ABB RAPID module: P454.mod

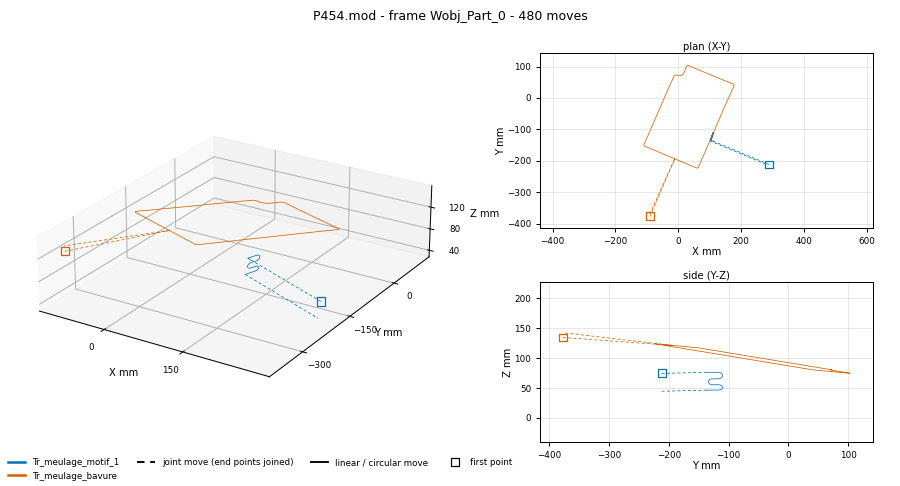
[picture p0: tool path of P454.mod in frame Wobj_Part_0, 480 of 487 moves have a stored position in this frame; points joined in program order, loops and branches not executed]
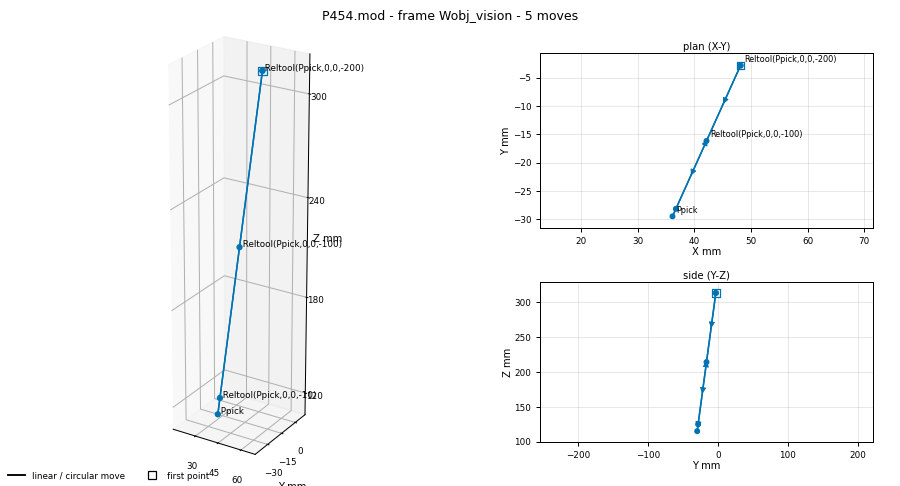
[picture p1: tool path of P454.mod in frame Wobj_vision, 5 of 487 moves have a stored position in this frame; points joined in program order, loops and branches not executed]
MODULE P454
	LOCAL CONST Speeddata vitesse_Tronconnage :=[10, 500, 0, 0];
	LOCAL CONST Robtarget Tr_meulage_motif_1_App1 :=[[289.653425414154,-211.82367493434,74.5113195582422],[0.591192296930468,-0.585574850342318,-0.390292937594222,0.394037035772936],[0,0,0,0],[8.999999E+09,8.999999E+09,8.999999E+09,8.999999E+09,8.999999E+09,8.999999E+09]];
	LOCAL CONST Robtarget Tr_meulage_motif_1_App2 :=[[114.292409942583,-138.712636871717,76.3252562122871],[0.591192296930468,-0.585574850342318,-0.390292937594222,0.394037035772936],[0,0,0,0],[8.999999E+09,8.999999E+09,8.999999E+09,8.999999E+09,8.999999E+09,8.999999E+09]];
	LOCAL CONST Robtarget Tr_meulage_motif_1_P0 :=[[105.0628828125,-134.8646875,76.4207265625],[0.591192296930468,-0.585574850342318,-0.390292937594222,0.394037035772936],[0,0,0,0],[8.999999E+09,8.999999E+09,8.999999E+09,8.999999E+09,8.999999E+09,8.999999E+09]];
	LOCAL CONST Robtarget Tr_meulage_motif_1_P1 :=[[105.3932265625,-133.920828125,76.423703125],[0.591192296930468,-0.585574850342318,-0.390292937594222,0.394037035772936],[0,0,0,0],[8.999999E+09,8.999999E+09,8.999999E+09,8.999999E+09,8.999999E+09,8.999999E+09]];
	LOCAL CONST Robtarget Tr_meulage_motif_1_P2 :=[[105.7235703125,-132.97696875,76.426671875],[0.591192296930468,-0.585574850342318,-0.390292937594222,0.394037035772936],[0,0,0,0],[8.999999E+09,8.999999E+09,8.999999E+09,8.999999E+09,8.999999E+09,8.999999E+09]];
	LOCAL CONST Robtarget Tr_meulage_motif_1_P3 :=[[106.0539140625,-132.033109375,76.4296484375],[0.591192296930468,-0.585574850342318,-0.390292937594222,0.394037035772936],[0,0,0,0],[8.999999E+09,8.999999E+09,8.999999E+09,8.999999E+09,8.999999E+09,8.999999E+09]];
	LOCAL CONST Robtarget Tr_meulage_motif_1_P4 :=[[106.3842578125,-131.089265625,76.4326171875],[0.591192296930468,-0.585574850342318,-0.390292937594222,0.394037035772936],[0,0,0,0],[8.999999E+09,8.999999E+09,8.999999E+09,8.999999E+09,8.999999E+09,8.999999E+09]];
	LOCAL CONST Robtarget Tr_meulage_motif_1_P5 :=[[106.7146015625,-130.14540625,76.43559375],[0.591192296930468,-0.585574850342318,-0.390292937594222,0.394037035772936],[0,0,0,0],[8.999999E+09,8.999999E+09,8.999999E+09,8.999999E+09,8.999999E+09,8.999999E+09]];
	LOCAL CONST Robtarget Tr_meulage_motif_1_P6 :=[[107.0449453125,-129.201546875,76.4385625],[0.591192296930468,-0.585574850342318,-0.390292937594222,0.394037035772936],[0,0,0,0],[8.999999E+09,8.999999E+09,8.999999E+09,8.999999E+09,8.999999E+09,8.999999E+09]];
	LOCAL CONST Robtarget Tr_meulage_motif_1_P7 :=[[107.37528125,-128.2576953125,76.4415390625],[0.591192296930468,-0.585574850342318,-0.390292937594222,0.394037035772936],[0,0,0,0],[8.999999E+09,8.999999E+09,8.999999E+09,8.999999E+09,8.999999E+09,8.999999E+09]];
	LOCAL CONST Robtarget Tr_meulage_motif_1_P8 :=[[107.705625,-127.3138359375,76.4445078125],[0.591192296930468,-0.585574850342318,-0.390292937594222,0.394037035772936],[0,0,0,0],[8.999999E+09,8.999999E+09,8.999999E+09,8.999999E+09,8.999999E+09,8.999999E+09]];
	LOCAL CONST Robtarget Tr_meulage_motif_1_P9 :=[[108.03596875,-126.3699765625,76.447484375],[0.591192296930468,-0.585574850342318,-0.390292937594222,0.394037035772936],[0,0,0,0],[8.999999E+09,8.999999E+09,8.999999E+09,8.999999E+09,8.999999E+09,8.999999E+09]];
	LOCAL CONST Robtarget Tr_meulage_motif_1_P10 :=[[108.3663125,-125.426125,76.450453125],[0.591192296930468,-0.585574850342318,-0.390292937594222,0.394037035772936],[0,0,0,0],[8.999999E+09,8.999999E+09,8.999999E+09,8.999999E+09,8.999999E+09,8.999999E+09]];
	LOCAL CONST Robtarget Tr_meulage_motif_1_P11 :=[[108.69665625,-124.482265625,76.4534296875],[0.591192296930468,-0.585574850342318,-0.390292937594222,0.394037035772936],[0,0,0,0],[8.999999E+09,8.999999E+09,8.999999E+09,8.999999E+09,8.999999E+09,8.999999E+09]];
	LOCAL CONST Robtarget Tr_meulage_motif_1_P12 :=[[109.027,-123.5384140625,76.4563984375],[0.591192296930468,-0.585574850342318,-0.390292937594222,0.394037035772936],[0,0,0,0],[8.999999E+09,8.999999E+09,8.999999E+09,8.999999E+09,8.999999E+09,8.999999E+09]];
	LOCAL CONST Robtarget Tr_meulage_motif_1_P13 :=[[109.35734375,-122.5945546875,76.459375],[0.591192296930468,-0.585574850342318,-0.390292937594222,0.394037035772936],[0,0,0,0],[8.999999E+09,8.999999E+09,8.999999E+09,8.999999E+09,8.999999E+09,8.999999E+09]];
	LOCAL CONST Robtarget Tr_meulage_motif_1_P14 :=[[109.6876875,-121.6506953125,76.46234375],[0.591192296930468,-0.585574850342318,-0.390292937594222,0.394037035772936],[0,0,0,0],[8.999999E+09,8.999999E+09,8.999999E+09,8.999999E+09,8.999999E+09,8.999999E+09]];
	LOCAL CONST Robtarget Tr_meulage_motif_1_P15 :=[[110.01803125,-120.70684375,76.4653203125],[0.591192296930468,-0.585574850342318,-0.390292937594222,0.394037035772936],[0,0,0,0],[8.999999E+09,8.999999E+09,8.999999E+09,8.999999E+09,8.999999E+09,8.999999E+09]];
	LOCAL CONST Robtarget Tr_meulage_motif_1_P16 :=[[110.348375,-119.762984375,76.4682890625],[0.591192296930468,-0.585574850342318,-0.390292937594222,0.394037035772936],[0,0,0,0],[8.999999E+09,8.999999E+09,8.999999E+09,8.999999E+09,8.999999E+09,8.999999E+09]];
	LOCAL CONST Robtarget Tr_meulage_motif_1_P17 :=[[110.67871875,-118.8191328125,76.471265625],[0.591192296930468,-0.585574850342318,-0.390292937594222,0.394037035772936],[0,0,0,0],[8.999999E+09,8.999999E+09,8.999999E+09,8.999999E+09,8.999999E+09,8.999999E+09]];
	LOCAL CONST Robtarget Tr_meulage_motif_1_P18 :=[[111.0090625,-117.8752734375,76.474234375],[0.591192296930468,-0.585574850342318,-0.390292937594222,0.394037035772936],[0,0,0,0],[8.999999E+09,8.999999E+09,8.999999E+09,8.999999E+09,8.999999E+09,8.999999E+09]];
	LOCAL CONST Robtarget Tr_meulage_motif_1_P19 :=[[111.33940625,-116.931421875,76.4772109375],[0.591192296930468,-0.585574850342318,-0.390292937594222,0.394037035772936],[0,0,0,0],[8.999999E+09,8.999999E+09,8.999999E+09,8.999999E+09,8.999999E+09,8.999999E+09]];
	LOCAL CONST Robtarget Tr_meulage_motif_1_P20 :=[[111.6568125,-115.9905703125,76.370140625],[0.591192296930468,-0.585574850342318,-0.390292937594222,0.394037035772936],[0,0,0,0],[8.999999E+09,8.999999E+09,8.999999E+09,8.999999E+09,8.999999E+09,8.999999E+09]];
	LOCAL CONST Robtarget Tr_meulage_motif_1_P21 :=[[111.9494609375,-115.0895390625,76.1628515625],[0.591192296930468,-0.585574850342318,-0.390292937594222,0.394037035772936],[0,0,0,0],[8.999999E+09,8.999999E+09,8.999999E+09,8.999999E+09,8.999999E+09,8.999999E+09]];
	LOCAL CONST Robtarget Tr_meulage_motif_1_P22 :=[[112.2053828125,-114.274828125,75.894953125],[0.591192296930468,-0.585574850342318,-0.390292937594222,0.394037035772936],[0,0,0,0],[8.999999E+09,8.999999E+09,8.999999E+09,8.999999E+09,8.999999E+09,8.999999E+09]];
	LOCAL CONST Robtarget Tr_meulage_motif_1_P23 :=[[112.42696875,-113.5569765625,75.6226640625],[0.591192296930468,-0.585574850342318,-0.390292937594222,0.394037035772936],[0,0,0,0],[8.999999E+09,8.999999E+09,8.999999E+09,8.999999E+09,8.999999E+09,8.999999E+09]];
	LOCAL CONST Robtarget Tr_meulage_motif_1_P24 :=[[112.732296875,-112.495359375,75.013],[0.591192296930468,-0.585574850342318,-0.390292937594222,0.394037035772936],[0,0,0,0],[8.999999E+09,8.999999E+09,8.999999E+09,8.999999E+09,8.999999E+09,8.999999E+09]];
	LOCAL CONST Robtarget Tr_meulage_motif_1_P25 :=[[112.9901796875,-111.4981875,74.172765625],[0.591192296930468,-0.585574850342318,-0.390292937594222,0.394037035772936],[0,0,0,0],[8.999999E+09,8.999999E+09,8.999999E+09,8.999999E+09,8.999999E+09,8.999999E+09]];
	LOCAL CONST Robtarget Tr_meulage_motif_1_P26 :=[[113.1731484375,-110.660953125,73.1566953125],[0.591192296930468,-0.585574850342318,-0.390292937594222,0.394037035772936],[0,0,0,0],[8.999999E+09,8.999999E+09,8.999999E+09,8.999999E+09,8.999999E+09,8.999999E+09]];
	LOCAL CONST Robtarget Tr_meulage_motif_1_P27 :=[[113.228609375,-110.159671875,72.0477265625],[0.591192296930468,-0.585574850342318,-0.390292937594222,0.394037035772936],[0,0,0,0],[8.999999E+09,8.999999E+09,8.999999E+09,8.999999E+09,8.999999E+09,8.999999E+09]];
	LOCAL CONST Robtarget Tr_meulage_motif_1_P28 :=[[113.171578125,-110.108859375,71.3554296875],[0.591192296930468,-0.585574850342318,-0.390292937594222,0.394037035772936],[0,0,0,0],[8.999999E+09,8.999999E+09,8.999999E+09,8.999999E+09,8.999999E+09,8.999999E+09]];
	LOCAL CONST Robtarget Tr_meulage_motif_1_P29 :=[[113.1088984375,-110.0848515625,70.69759375],[0.591192296930468,-0.585574850342318,-0.390292937594222,0.394037035772936],[0,0,0,0],[8.999999E+09,8.999999E+09,8.999999E+09,8.999999E+09,8.999999E+09,8.999999E+09]];
	LOCAL CONST Robtarget Tr_meulage_motif_1_P30 :=[[113.028109375,-110.1126484375,70.03975],[0.591192296930468,-0.585574850342318,-0.390292937594222,0.394037035772936],[0,0,0,0],[8.999999E+09,8.999999E+09,8.999999E+09,8.999999E+09,8.999999E+09,8.999999E+09]];
	LOCAL CONST Robtarget Tr_meulage_motif_1_P31 :=[[112.75909375,-110.542890625,68.9422109375],[0.591192296930468,-0.585574850342318,-0.390292937594222,0.394037035772936],[0,0,0,0],[8.999999E+09,8.999999E+09,8.999999E+09,8.999999E+09,8.999999E+09,8.999999E+09]];
	LOCAL CONST Robtarget Tr_meulage_motif_1_P32 :=[[112.3806953125,-111.314875,67.9382421875],[0.591192296930468,-0.585574850342318,-0.390292937594222,0.394037035772936],[0,0,0,0],[8.999999E+09,8.999999E+09,8.999999E+09,8.999999E+09,8.999999E+09,8.999999E+09]];
	LOCAL CONST Robtarget Tr_meulage_motif_1_P33 :=[[111.9640546875,-112.2507265625,67.1106015625],[0.591192296930468,-0.585574850342318,-0.390292937594222,0.394037035772936],[0,0,0,0],[8.999999E+09,8.999999E+09,8.999999E+09,8.999999E+09,8.999999E+09,8.999999E+09]];
	LOCAL CONST Robtarget Tr_meulage_motif_1_P34 :=[[111.6995703125,-112.884875,66.7148515625],[0.591192296930468,-0.585574850342318,-0.390292937594222,0.394037035772936],[0,0,0,0],[8.999999E+09,8.999999E+09,8.999999E+09,8.999999E+09,8.999999E+09,8.999999E+09]];
	LOCAL CONST Robtarget Tr_meulage_motif_1_P35 :=[[111.270765625,-113.9603046875,66.2263984375],[0.591192296930468,-0.585574850342318,-0.390292937594222,0.394037035772936],[0,0,0,0],[8.999999E+09,8.999999E+09,8.999999E+09,8.999999E+09,8.999999E+09,8.999999E+09]];
	LOCAL CONST Robtarget Tr_meulage_motif_1_P36 :=[[110.9665859375,-114.7483046875,65.96115625],[0.591192296930468,-0.585574850342318,-0.390292937594222,0.394037035772936],[0,0,0,0],[8.999999E+09,8.999999E+09,8.999999E+09,8.999999E+09,8.999999E+09,8.999999E+09]];
	LOCAL CONST Robtarget Tr_meulage_motif_1_P37 :=[[110.6393203125,-115.6205546875,65.7549765625],[0.591192296930468,-0.585574850342318,-0.390292937594222,0.394037035772936],[0,0,0,0],[8.999999E+09,8.999999E+09,8.999999E+09,8.999999E+09,8.999999E+09,8.999999E+09]];
	LOCAL CONST Robtarget Tr_meulage_motif_1_P38 :=[[110.3047734375,-116.5430625,65.6440234375],[0.591192296930468,-0.585574850342318,-0.390292937594222,0.394037035772936],[0,0,0,0],[8.999999E+09,8.999999E+09,8.999999E+09,8.999999E+09,8.999999E+09,8.999999E+09]];
	LOCAL CONST Robtarget Tr_meulage_motif_1_P39 :=[[109.96640625,-117.4758828125,65.53105078125],[0.591192296930468,-0.585574850342318,-0.390292937594222,0.394037035772936],[0,0,0,0],[8.999999E+09,8.999999E+09,8.999999E+09,8.999999E+09,8.999999E+09,8.999999E+09]];
	LOCAL CONST Robtarget Tr_meulage_motif_1_P40 :=[[109.6360625,-118.4197421875,65.528078125],[0.591192296930468,-0.585574850342318,-0.390292937594222,0.394037035772936],[0,0,0,0],[8.999999E+09,8.999999E+09,8.999999E+09,8.999999E+09,8.999999E+09,8.999999E+09]];
	LOCAL CONST Robtarget Tr_meulage_motif_1_P41 :=[[109.30571875,-119.3636015625,65.52510546875],[0.591192296930468,-0.585574850342318,-0.390292937594222,0.394037035772936],[0,0,0,0],[8.999999E+09,8.999999E+09,8.999999E+09,8.999999E+09,8.999999E+09,8.999999E+09]];
	LOCAL CONST Robtarget Tr_meulage_motif_1_P42 :=[[108.975375,-120.307453125,65.5221328125],[0.591192296930468,-0.585574850342318,-0.390292937594222,0.394037035772936],[0,0,0,0],[8.999999E+09,8.999999E+09,8.999999E+09,8.999999E+09,8.999999E+09,8.999999E+09]];
	LOCAL CONST Robtarget Tr_meulage_motif_1_P43 :=[[108.64503125,-121.2513125,65.51916015625],[0.591192296930468,-0.585574850342318,-0.390292937594222,0.394037035772936],[0,0,0,0],[8.999999E+09,8.999999E+09,8.999999E+09,8.999999E+09,8.999999E+09,8.999999E+09]];
	LOCAL CONST Robtarget Tr_meulage_motif_1_P44 :=[[108.3146875,-122.1951640625,65.5161875],[0.591192296930468,-0.585574850342318,-0.390292937594222,0.394037035772936],[0,0,0,0],[8.999999E+09,8.999999E+09,8.999999E+09,8.999999E+09,8.999999E+09,8.999999E+09]];
	LOCAL CONST Robtarget Tr_meulage_motif_1_P45 :=[[107.98434375,-123.1390234375,65.51321484375],[0.591192296930468,-0.585574850342318,-0.390292937594222,0.394037035772936],[0,0,0,0],[8.999999E+09,8.999999E+09,8.999999E+09,8.999999E+09,8.999999E+09,8.999999E+09]];
	LOCAL CONST Robtarget Tr_meulage_motif_1_P46 :=[[107.654,-124.0828828125,65.5102421875],[0.591192296930468,-0.585574850342318,-0.390292937594222,0.394037035772936],[0,0,0,0],[8.999999E+09,8.999999E+09,8.999999E+09,8.999999E+09,8.999999E+09,8.999999E+09]];
	LOCAL CONST Robtarget Tr_meulage_motif_1_P47 :=[[107.32365625,-125.026734375,65.50726953125],[0.591192296930468,-0.585574850342318,-0.390292937594222,0.394037035772936],[0,0,0,0],[8.999999E+09,8.999999E+09,8.999999E+09,8.999999E+09,8.999999E+09,8.999999E+09]];
	LOCAL CONST Robtarget Tr_meulage_motif_1_P48 :=[[106.9933125,-125.97059375,65.504296875],[0.591192296930468,-0.585574850342318,-0.390292937594222,0.394037035772936],[0,0,0,0],[8.999999E+09,8.999999E+09,8.999999E+09,8.999999E+09,8.999999E+09,8.999999E+09]];
	LOCAL CONST Robtarget Tr_meulage_motif_1_P49 :=[[106.66296875,-126.9144453125,65.50132421875],[0.591192296930468,-0.585574850342318,-0.390292937594222,0.394037035772936],[0,0,0,0],[8.999999E+09,8.999999E+09,8.999999E+09,8.999999E+09,8.999999E+09,8.999999E+09]];
	LOCAL CONST Robtarget Tr_meulage_motif_1_P50 :=[[106.332625,-127.8583046875,65.4983515625],[0.591192296930468,-0.585574850342318,-0.390292937594222,0.394037035772936],[0,0,0,0],[8.999999E+09,8.999999E+09,8.999999E+09,8.999999E+09,8.999999E+09,8.999999E+09]];
	LOCAL CONST Robtarget Tr_meulage_motif_1_P51 :=[[105.9942578125,-128.791125,65.385375],[0.591192296930468,-0.585574850342318,-0.390292937594222,0.394037035772936],[0,0,0,0],[8.999999E+09,8.999999E+09,8.999999E+09,8.999999E+09,8.999999E+09,8.999999E+09]];
	LOCAL CONST Robtarget Tr_meulage_motif_1_P52 :=[[105.6615703125,-129.6768125,65.17246484375],[0.591192296930468,-0.585574850342318,-0.390292937594222,0.394037035772936],[0,0,0,0],[8.999999E+09,8.999999E+09,8.999999E+09,8.999999E+09,8.999999E+09,8.999999E+09]];
	LOCAL CONST Robtarget Tr_meulage_motif_1_P53 :=[[105.3541171875,-130.4717890625,64.8994921875],[0.591192296930468,-0.585574850342318,-0.390292937594222,0.394037035772936],[0,0,0,0],[8.999999E+09,8.999999E+09,8.999999E+09,8.999999E+09,8.999999E+09,8.999999E+09]];
	LOCAL CONST Robtarget Tr_meulage_motif_1_P54 :=[[105.0902421875,-131.132296875,64.59479296875],[0.591192296930468,-0.585574850342318,-0.390292937594222,0.394037035772936],[0,0,0,0],[8.999999E+09,8.999999E+09,8.999999E+09,8.999999E+09,8.999999E+09,8.999999E+09]];
	LOCAL CONST Robtarget Tr_meulage_motif_1_P55 :=[[104.6857109375,-132.084640625,63.93260546875],[0.591192296930468,-0.585574850342318,-0.390292937594222,0.394037035772936],[0,0,0,0],[8.999999E+09,8.999999E+09,8.999999E+09,8.999999E+09,8.999999E+09,8.999999E+09]];
	LOCAL CONST Robtarget Tr_meulage_motif_1_P56 :=[[104.3022734375,-132.9031875,63.03264453125],[0.591192296930468,-0.585574850342318,-0.390292937594222,0.394037035772936],[0,0,0,0],[8.999999E+09,8.999999E+09,8.999999E+09,8.999999E+09,8.999999E+09,8.999999E+09]];
	LOCAL CONST Robtarget Tr_meulage_motif_1_P57 :=[[104.0263984375,-133.370140625,61.99042578125],[0.591192296930468,-0.585574850342318,-0.390292937594222,0.394037035772936],[0,0,0,0],[8.999999E+09,8.999999E+09,8.999999E+09,8.999999E+09,8.999999E+09,8.999999E+09]];
	LOCAL CONST Robtarget Tr_meulage_motif_1_P58 :=[[103.8996484375,-133.519375,61.30023828125],[0.591192296930468,-0.585574850342318,-0.390292937594222,0.394037035772936],[0,0,0,0],[8.999999E+09,8.999999E+09,8.999999E+09,8.999999E+09,8.999999E+09,8.999999E+09]];
	LOCAL CONST Robtarget Tr_meulage_motif_1_P59 :=[[103.805578125,-133.5516875,60.53402734375],[0.591192296930468,-0.585574850342318,-0.390292937594222,0.394037035772936],[0,0,0,0],[8.999999E+09,8.999999E+09,8.999999E+09,8.999999E+09,8.999999E+09,8.999999E+09]];
	LOCAL CONST Robtarget Tr_meulage_motif_1_P60 :=[[103.7547109375,-133.460546875,59.768328125],[0.591192296930468,-0.585574850342318,-0.390292937594222,0.394037035772936],[0,0,0,0],[8.999999E+09,8.999999E+09,8.999999E+09,8.999999E+09,8.999999E+09,8.999999E+09]];
	LOCAL CONST Robtarget Tr_meulage_motif_1_P61 :=[[103.7882734375,-133.024265625,58.667046875],[0.591192296930468,-0.585574850342318,-0.390292937594222,0.394037035772936],[0,0,0,0],[8.999999E+09,8.999999E+09,8.999999E+09,8.999999E+09,8.999999E+09,8.999999E+09]];
	LOCAL CONST Robtarget Tr_meulage_motif_1_P62 :=[[103.869625,-132.611953125,58.0856171875],[0.591192296930468,-0.585574850342318,-0.390292937594222,0.394037035772936],[0,0,0,0],[8.999999E+09,8.999999E+09,8.999999E+09,8.999999E+09,8.999999E+09,8.999999E+09]];
	LOCAL CONST Robtarget Tr_meulage_motif_1_P63 :=[[104.07859375,-131.742421875,57.2057109375],[0.591192296930468,-0.585574850342318,-0.390292937594222,0.394037035772936],[0,0,0,0],[8.999999E+09,8.999999E+09,8.999999E+09,8.999999E+09,8.999999E+09,8.999999E+09]];
	LOCAL CONST Robtarget Tr_meulage_motif_1_P64 :=[[104.232796875,-131.174578125,56.79528125],[0.591192296930468,-0.585574850342318,-0.390292937594222,0.394037035772936],[0,0,0,0],[8.999999E+09,8.999999E+09,8.999999E+09,8.999999E+09,8.999999E+09,8.999999E+09]];
	LOCAL CONST Robtarget Tr_meulage_motif_1_P65 :=[[104.550515625,-130.0996796875,56.2573203125],[0.591192296930468,-0.585574850342318,-0.390292937594222,0.394037035772936],[0,0,0,0],[8.999999E+09,8.999999E+09,8.999999E+09,8.999999E+09,8.999999E+09,8.999999E+09]];
	LOCAL CONST Robtarget Tr_meulage_motif_1_P66 :=[[104.7952421875,-129.3097109375,55.96580078125],[0.591192296930468,-0.585574850342318,-0.390292937594222,0.394037035772936],[0,0,0,0],[8.999999E+09,8.999999E+09,8.999999E+09,8.999999E+09,8.999999E+09,8.999999E+09]];
	LOCAL CONST Robtarget Tr_meulage_motif_1_P67 :=[[105.0837421875,-128.4226171875,55.76515625],[0.591192296930468,-0.585574850342318,-0.390292937594222,0.394037035772936],[0,0,0,0],[8.999999E+09,8.999999E+09,8.999999E+09,8.999999E+09,8.999999E+09,8.999999E+09]];
	LOCAL CONST Robtarget Tr_meulage_motif_1_P68 :=[[105.3976953125,-127.49221875,55.66004296875],[0.591192296930468,-0.585574850342318,-0.390292937594222,0.394037035772936],[0,0,0,0],[8.999999E+09,8.999999E+09,8.999999E+09,8.999999E+09,8.999999E+09,8.999999E+09]];
	LOCAL CONST Robtarget Tr_meulage_motif_1_P69 :=[[105.7151015625,-126.5513671875,55.55296875],[0.591192296930468,-0.585574850342318,-0.390292937594222,0.394037035772936],[0,0,0,0],[8.999999E+09,8.999999E+09,8.999999E+09,8.999999E+09,8.999999E+09,8.999999E+09]];
	LOCAL CONST Robtarget Tr_meulage_motif_1_P70 :=[[106.0454453125,-125.6075078125,55.55594140625],[0.591192296930468,-0.585574850342318,-0.390292937594222,0.394037035772936],[0,0,0,0],[8.999999E+09,8.999999E+09,8.999999E+09,8.999999E+09,8.999999E+09,8.999999E+09]];
	LOCAL CONST Robtarget Tr_meulage_motif_1_P71 :=[[106.3757890625,-124.66365625,55.5589140625],[0.591192296930468,-0.585574850342318,-0.390292937594222,0.394037035772936],[0,0,0,0],[8.999999E+09,8.999999E+09,8.999999E+09,8.999999E+09,8.999999E+09,8.999999E+09]];
	LOCAL CONST Robtarget Tr_meulage_motif_1_P72 :=[[106.7061328125,-123.719796875,55.56188671875],[0.591192296930468,-0.585574850342318,-0.390292937594222,0.394037035772936],[0,0,0,0],[8.999999E+09,8.999999E+09,8.999999E+09,8.999999E+09,8.999999E+09,8.999999E+09]];
	LOCAL CONST Robtarget Tr_meulage_motif_1_P73 :=[[107.0364765625,-122.7759453125,55.564859375],[0.591192296930468,-0.585574850342318,-0.390292937594222,0.394037035772936],[0,0,0,0],[8.999999E+09,8.999999E+09,8.999999E+09,8.999999E+09,8.999999E+09,8.999999E+09]];
	LOCAL CONST Robtarget Tr_meulage_motif_1_P74 :=[[107.3668203125,-121.8320859375,55.56783203125],[0.591192296930468,-0.585574850342318,-0.390292937594222,0.394037035772936],[0,0,0,0],[8.999999E+09,8.999999E+09,8.999999E+09,8.999999E+09,8.999999E+09,8.999999E+09]];
	LOCAL CONST Robtarget Tr_meulage_motif_1_P75 :=[[107.6971640625,-120.8882265625,55.5708046875],[0.591192296930468,-0.585574850342318,-0.390292937594222,0.394037035772936],[0,0,0,0],[8.999999E+09,8.999999E+09,8.999999E+09,8.999999E+09,8.999999E+09,8.999999E+09]];
	LOCAL CONST Robtarget Tr_meulage_motif_1_P76 :=[[108.0275078125,-119.944375,55.57377734375],[0.591192296930468,-0.585574850342318,-0.390292937594222,0.394037035772936],[0,0,0,0],[8.999999E+09,8.999999E+09,8.999999E+09,8.999999E+09,8.999999E+09,8.999999E+09]];
	LOCAL CONST Robtarget Tr_meulage_motif_1_P77 :=[[108.3578515625,-119.000515625,55.57675],[0.591192296930468,-0.585574850342318,-0.390292937594222,0.394037035772936],[0,0,0,0],[8.999999E+09,8.999999E+09,8.999999E+09,8.999999E+09,8.999999E+09,8.999999E+09]];
	LOCAL CONST Robtarget Tr_meulage_motif_1_P78 :=[[108.6881953125,-118.0566640625,55.57972265625],[0.591192296930468,-0.585574850342318,-0.390292937594222,0.394037035772936],[0,0,0,0],[8.999999E+09,8.999999E+09,8.999999E+09,8.999999E+09,8.999999E+09,8.999999E+09]];
	LOCAL CONST Robtarget Tr_meulage_motif_1_P79 :=[[109.0185390625,-117.1128046875,55.5826953125],[0.591192296930468,-0.585574850342318,-0.390292937594222,0.394037035772936],[0,0,0,0],[8.999999E+09,8.999999E+09,8.999999E+09,8.999999E+09,8.999999E+09,8.999999E+09]];
	LOCAL CONST Robtarget Tr_meulage_motif_1_P80 :=[[109.3488828125,-116.168953125,55.58566796875],[0.591192296930468,-0.585574850342318,-0.390292937594222,0.394037035772936],[0,0,0,0],[8.999999E+09,8.999999E+09,8.999999E+09,8.999999E+09,8.999999E+09,8.999999E+09]];
	LOCAL CONST Robtarget Tr_meulage_motif_1_P81 :=[[109.66628125,-115.2281015625,55.47859765625],[0.591192296930468,-0.585574850342318,-0.390292937594222,0.394037035772936],[0,0,0,0],[8.999999E+09,8.999999E+09,8.999999E+09,8.999999E+09,8.999999E+09,8.999999E+09]];
	LOCAL CONST Robtarget Tr_meulage_motif_1_P82 :=[[109.9589375,-114.3270703125,55.2713125],[0.591192296930468,-0.585574850342318,-0.390292937594222,0.394037035772936],[0,0,0,0],[8.999999E+09,8.999999E+09,8.999999E+09,8.999999E+09,8.999999E+09,8.999999E+09]];
	LOCAL CONST Robtarget Tr_meulage_motif_1_P83 :=[[110.214859375,-113.512359375,55.00341015625],[0.591192296930468,-0.585574850342318,-0.390292937594222,0.394037035772936],[0,0,0,0],[8.999999E+09,8.999999E+09,8.999999E+09,8.999999E+09,8.999999E+09,8.999999E+09]];
	LOCAL CONST Robtarget Tr_meulage_motif_1_P84 :=[[110.4364375,-112.7945078125,54.731125],[0.591192296930468,-0.585574850342318,-0.390292937594222,0.394037035772936],[0,0,0,0],[8.999999E+09,8.999999E+09,8.999999E+09,8.999999E+09,8.999999E+09,8.999999E+09]];
	LOCAL CONST Robtarget Tr_meulage_motif_1_P85 :=[[110.741765625,-111.732890625,54.12145703125],[0.591192296930468,-0.585574850342318,-0.390292937594222,0.394037035772936],[0,0,0,0],[8.999999E+09,8.999999E+09,8.999999E+09,8.999999E+09,8.999999E+09,8.999999E+09]];
	LOCAL CONST Robtarget Tr_meulage_motif_1_P86 :=[[110.99965625,-110.73571875,53.28122265625],[0.591192296930468,-0.585574850342318,-0.390292937594222,0.394037035772936],[0,0,0,0],[8.999999E+09,8.999999E+09,8.999999E+09,8.999999E+09,8.999999E+09,8.999999E+09]];
	LOCAL CONST Robtarget Tr_meulage_motif_1_P87 :=[[111.1472734375,-109.9868671875,52.22401953125],[0.591192296930468,-0.585574850342318,-0.390292937594222,0.394037035772936],[0,0,0,0],[8.999999E+09,8.999999E+09,8.999999E+09,8.999999E+09,8.999999E+09,8.999999E+09]];
	LOCAL CONST Robtarget Tr_meulage_motif_1_P88 :=[[111.175828125,-109.5640234375,51.11990234375],[0.591192296930468,-0.585574850342318,-0.390292937594222,0.394037035772936],[0,0,0,0],[8.999999E+09,8.999999E+09,8.999999E+09,8.999999E+09,8.999999E+09,8.999999E+09]];
	LOCAL CONST Robtarget Tr_meulage_motif_1_P89 :=[[111.0757578125,-109.67290625,50.546],[0.591192296930468,-0.585574850342318,-0.390292937594222,0.394037035772936],[0,0,0,0],[8.999999E+09,8.999999E+09,8.999999E+09,8.999999E+09,8.999999E+09,8.999999E+09]];
	LOCAL CONST Robtarget Tr_meulage_motif_1_P90 :=[[111.0245390625,-109.7222265625,50.23159765625],[0.591192296930468,-0.585574850342318,-0.390292937594222,0.394037035772936],[0,0,0,0],[8.999999E+09,8.999999E+09,8.999999E+09,8.999999E+09,8.999999E+09,8.999999E+09]];
	LOCAL CONST Robtarget Tr_meulage_motif_1_P91 :=[[110.8130078125,-110.0474453125,49.3261953125],[0.591192296930468,-0.585574850342318,-0.390292937594222,0.394037035772936],[0,0,0,0],[8.999999E+09,8.999999E+09,8.999999E+09,8.999999E+09,8.999999E+09,8.999999E+09]];
	LOCAL CONST Robtarget Tr_meulage_motif_1_P92 :=[[110.64378125,-110.3681328125,48.79767578125],[0.591192296930468,-0.585574850342318,-0.390292937594222,0.394037035772936],[0,0,0,0],[8.999999E+09,8.999999E+09,8.999999E+09,8.999999E+09,8.999999E+09,8.999999E+09]];
	LOCAL CONST Robtarget Tr_meulage_motif_1_P93 :=[[110.21025,-111.371140625,48.031046875],[0.591192296930468,-0.585574850342318,-0.390292937594222,0.394037035772936],[0,0,0,0],[8.999999E+09,8.999999E+09,8.999999E+09,8.999999E+09,8.999999E+09,8.999999E+09]];
	LOCAL CONST Robtarget Tr_meulage_motif_1_P94 :=[[109.9119609375,-112.1030625,47.63887890625],[0.591192296930468,-0.585574850342318,-0.390292937594222,0.394037035772936],[0,0,0,0],[8.999999E+09,8.999999E+09,8.999999E+09,8.999999E+09,8.999999E+09,8.999999E+09]];
	LOCAL CONST Robtarget Tr_meulage_motif_1_P95 :=[[109.486484375,-113.200609375,47.25276953125],[0.591192296930468,-0.585574850342318,-0.390292937594222,0.394037035772936],[0,0,0,0],[8.999999E+09,8.999999E+09,8.999999E+09,8.999999E+09,8.999999E+09,8.999999E+09]];
	LOCAL CONST Robtarget Tr_meulage_motif_1_P96 :=[[109.1656328125,-114.058453125,47.05928515625],[0.591192296930468,-0.585574850342318,-0.390292937594222,0.394037035772936],[0,0,0,0],[8.999999E+09,8.999999E+09,8.999999E+09,8.999999E+09,8.999999E+09,8.999999E+09]];
	LOCAL CONST Robtarget Tr_meulage_motif_1_P97 :=[[108.8383671875,-114.930703125,46.8531015625],[0.591192296930468,-0.585574850342318,-0.390292937594222,0.394037035772936],[0,0,0,0],[8.999999E+09,8.999999E+09,8.999999E+09,8.999999E+09,8.999999E+09,8.999999E+09]];
	LOCAL CONST Robtarget Tr_meulage_motif_1_P98 :=[[108.5038203125,-115.8532109375,46.74215234375],[0.591192296930468,-0.585574850342318,-0.390292937594222,0.394037035772936],[0,0,0,0],[8.999999E+09,8.999999E+09,8.999999E+09,8.999999E+09,8.999999E+09,8.999999E+09]];
	LOCAL CONST Robtarget Tr_meulage_motif_1_P99 :=[[108.165453125,-116.78603125,46.6291796875],[0.591192296930468,-0.585574850342318,-0.390292937594222,0.394037035772936],[0,0,0,0],[8.999999E+09,8.999999E+09,8.999999E+09,8.999999E+09,8.999999E+09,8.999999E+09]];
	LOCAL CONST Robtarget Tr_meulage_motif_1_P100 :=[[107.835109375,-117.729890625,46.62620703125],[0.591192296930468,-0.585574850342318,-0.390292937594222,0.394037035772936],[0,0,0,0],[8.999999E+09,8.999999E+09,8.999999E+09,8.999999E+09,8.999999E+09,8.999999E+09]];
	LOCAL CONST Robtarget Tr_meulage_motif_1_P101 :=[[107.504765625,-118.6737421875,46.623234375],[0.591192296930468,-0.585574850342318,-0.390292937594222,0.394037035772936],[0,0,0,0],[8.999999E+09,8.999999E+09,8.999999E+09,8.999999E+09,8.999999E+09,8.999999E+09]];
	LOCAL CONST Robtarget Tr_meulage_motif_1_P102 :=[[107.174421875,-119.6176015625,46.62026171875],[0.591192296930468,-0.585574850342318,-0.390292937594222,0.394037035772936],[0,0,0,0],[8.999999E+09,8.999999E+09,8.999999E+09,8.999999E+09,8.999999E+09,8.999999E+09]];
	LOCAL CONST Robtarget Tr_meulage_motif_1_P103 :=[[106.844078125,-120.5614609375,46.6172890625],[0.591192296930468,-0.585574850342318,-0.390292937594222,0.394037035772936],[0,0,0,0],[8.999999E+09,8.999999E+09,8.999999E+09,8.999999E+09,8.999999E+09,8.999999E+09]];
	LOCAL CONST Robtarget Tr_meulage_motif_1_P104 :=[[106.513734375,-121.5053125,46.61431640625],[0.591192296930468,-0.585574850342318,-0.390292937594222,0.394037035772936],[0,0,0,0],[8.999999E+09,8.999999E+09,8.999999E+09,8.999999E+09,8.999999E+09,8.999999E+09]];
	LOCAL CONST Robtarget Tr_meulage_motif_1_P105 :=[[106.183390625,-122.449171875,46.61134375],[0.591192296930468,-0.585574850342318,-0.390292937594222,0.394037035772936],[0,0,0,0],[8.999999E+09,8.999999E+09,8.999999E+09,8.999999E+09,8.999999E+09,8.999999E+09]];
	LOCAL CONST Robtarget Tr_meulage_motif_1_P106 :=[[105.853046875,-123.3930234375,46.60837109375],[0.591192296930468,-0.585574850342318,-0.390292937594222,0.394037035772936],[0,0,0,0],[8.999999E+09,8.999999E+09,8.999999E+09,8.999999E+09,8.999999E+09,8.999999E+09]];
	LOCAL CONST Robtarget Tr_meulage_motif_1_P107 :=[[105.522703125,-124.3368828125,46.6053984375],[0.591192296930468,-0.585574850342318,-0.390292937594222,0.394037035772936],[0,0,0,0],[8.999999E+09,8.999999E+09,8.999999E+09,8.999999E+09,8.999999E+09,8.999999E+09]];
	LOCAL CONST Robtarget Tr_meulage_motif_1_P108 :=[[105.192359375,-125.2807421875,46.60242578125],[0.591192296930468,-0.585574850342318,-0.390292937594222,0.394037035772936],[0,0,0,0],[8.999999E+09,8.999999E+09,8.999999E+09,8.999999E+09,8.999999E+09,8.999999E+09]];
	LOCAL CONST Robtarget Tr_meulage_motif_1_P109 :=[[104.862015625,-126.22459375,46.599453125],[0.591192296930468,-0.585574850342318,-0.390292937594222,0.394037035772936],[0,0,0,0],[8.999999E+09,8.999999E+09,8.999999E+09,8.999999E+09,8.999999E+09,8.999999E+09]];
	LOCAL CONST Robtarget Tr_meulage_motif_1_P110 :=[[104.531671875,-127.168453125,46.59648046875],[0.591192296930468,-0.585574850342318,-0.390292937594222,0.394037035772936],[0,0,0,0],[8.999999E+09,8.999999E+09,8.999999E+09,8.999999E+09,8.999999E+09,8.999999E+09]];
	LOCAL CONST Robtarget Tr_meulage_motif_1_P111 :=[[104.201328125,-128.1123046875,46.5935078125],[0.591192296930468,-0.585574850342318,-0.390292937594222,0.394037035772936],[0,0,0,0],[8.999999E+09,8.999999E+09,8.999999E+09,8.999999E+09,8.999999E+09,8.999999E+09]];
	LOCAL CONST Robtarget Tr_meulage_motif_1_P112 :=[[103.8709921875,-129.0561640625,46.59053515625],[0.591192296930468,-0.585574850342318,-0.390292937594222,0.394037035772936],[0,0,0,0],[8.999999E+09,8.999999E+09,8.999999E+09,8.999999E+09,8.999999E+09,8.999999E+09]];
	LOCAL CONST Robtarget Tr_meulage_motif_1_P113 :=[[103.5406484375,-130.000015625,46.5875625],[0.591192296930468,-0.585574850342318,-0.390292937594222,0.394037035772936],[0,0,0,0],[8.999999E+09,8.999999E+09,8.999999E+09,8.999999E+09,8.999999E+09,8.999999E+09]];
	LOCAL CONST Robtarget Tr_meulage_motif_1_P114 :=[[103.2103046875,-130.943875,46.58458984375],[0.591192296930468,-0.585574850342318,-0.390292937594222,0.394037035772936],[0,0,0,0],[8.999999E+09,8.999999E+09,8.999999E+09,8.999999E+09,8.999999E+09,8.999999E+09]];
	LOCAL CONST Robtarget Tr_meulage_motif_1_P115 :=[[102.8799609375,-131.887734375,46.5816171875],[0.591192296930468,-0.585574850342318,-0.390292937594222,0.394037035772936],[0,0,0,0],[8.999999E+09,8.999999E+09,8.999999E+09,8.999999E+09,8.999999E+09,8.999999E+09]];
	LOCAL CONST Robtarget Tr_meulage_motif_1_P116 :=[[102.5496171875,-132.83159375,46.57864453125],[0.591192296930468,-0.585574850342318,-0.390292937594222,0.394037035772936],[0,0,0,0],[8.999999E+09,8.999999E+09,8.999999E+09,8.999999E+09,8.999999E+09,8.999999E+09]];
	LOCAL CONST Robtarget Tr_meulage_motif_1_P117 :=[[102.2192734375,-133.7754375,46.575671875],[0.591192296930468,-0.585574850342318,-0.390292937594222,0.394037035772936],[0,0,0,0],[8.999999E+09,8.999999E+09,8.999999E+09,8.999999E+09,8.999999E+09,8.999999E+09]];
	LOCAL CONST Robtarget Tr_meulage_motif_1_P118 :=[[101.8889296875,-134.719296875,46.57269921875],[0.591192296930468,-0.585574850342318,-0.390292937594222,0.394037035772936],[0,0,0,0],[8.999999E+09,8.999999E+09,8.999999E+09,8.999999E+09,8.999999E+09,8.999999E+09]];
	LOCAL CONST Robtarget Tr_meulage_motif_1_P119 :=[[101.5585859375,-135.66315625,46.5697265625],[0.591192296930468,-0.585574850342318,-0.390292937594222,0.394037035772936],[0,0,0,0],[8.999999E+09,8.999999E+09,8.999999E+09,8.999999E+09,8.999999E+09,8.999999E+09]];
	LOCAL CONST Robtarget Tr_meulage_motif_1_P120 :=[[101.2282421875,-136.607015625,46.56675390625],[0.591192296930468,-0.585574850342318,-0.390292937594222,0.394037035772936],[0,0,0,0],[8.999999E+09,8.999999E+09,8.999999E+09,8.999999E+09,8.999999E+09,8.999999E+09]];
	LOCAL CONST Robtarget Tr_meulage_motif_1_degg1 :=[[110.457769317583,-140.454964996717,46.4712835560371],[0.591192296930468,-0.585574850342318,-0.390292937594222,0.394037035772936],[0,0,0,0],[8.999999E+09,8.999999E+09,8.999999E+09,8.999999E+09,8.999999E+09,8.999999E+09]];
	LOCAL CONST Robtarget Tr_meulage_motif_1_degg2 :=[[285.818784789154,-213.56600305934,44.6573469019922],[0.591192296930468,-0.585574850342318,-0.390292937594222,0.394037035772936],[0,0,0,0],[8.999999E+09,8.999999E+09,8.999999E+09,8.999999E+09,8.999999E+09,8.999999E+09]];
	LOCAL CONST Robtarget Tr_meulage_bavure_App1 :=[[-89.6194032030978,-377.065529328559,134.723885432184],[0.669210474743123,-0.715256266690532,0.147073413247032,-0.137605321735297],[0,0,0,0],[8.999999E+09,8.999999E+09,8.999999E+09,8.999999E+09,8.999999E+09,8.999999E+09]];
	LOCAL CONST Robtarget Tr_meulage_bavure_App2 :=[[-14.817870990233,-202.866346778928,122.099481380984],[0.669210474743123,-0.715256266690532,0.147073413247032,-0.137605321735297],[0,0,0,0],[8.999999E+09,8.999999E+09,8.999999E+09,8.999999E+09,8.999999E+09,8.999999E+09]];
	LOCAL CONST Robtarget Tr_meulage_bavure_P0 :=[[-10.8809482421875,-193.69796875,121.4350390625],[0.669210474743123,-0.715256266690532,0.147073413247032,-0.137605321735297],[0,0,0,0],[8.999999E+09,8.999999E+09,8.999999E+09,8.999999E+09,8.999999E+09,8.999999E+09]];
	LOCAL CONST Robtarget Tr_meulage_bavure_P1 :=[[-13.8624638671875,-192.46565625,121.324484375],[0.669223658494821,-0.715239070606633,0.147083014300852,-0.137620324417369],[0,0,0,0],[8.999999E+09,8.999999E+09,8.999999E+09,8.999999E+09,8.999999E+09,8.999999E+09]];
	LOCAL CONST Robtarget Tr_meulage_bavure_P2 :=[[-16.865427734375,-191.22528125,121.21325],[0.669258599663046,-0.715193827921842,0.147107614005423,-0.137659235727912],[0,0,0,0],[8.999999E+09,8.999999E+09,8.999999E+09,8.999999E+09,8.999999E+09,8.999999E+09]];
	LOCAL CONST Robtarget Tr_meulage_bavure_P3 :=[[-20.9573515625,-189.53415625,121.06153125],[0.669320704435918,-0.715118739396724,0.147137994316313,-0.137714900448788],[0,0,0,0],[8.999999E+09,8.999999E+09,8.999999E+09,8.999999E+09,8.999999E+09,8.999999E+09]];
	LOCAL CONST Robtarget Tr_meulage_bavure_P4 :=[[-24.6506796875,-187.945609375,120.915078125],[0.669405837354965,-0.715022181827208,0.147163657552376,-0.137775042391446],[0,0,0,0],[8.999999E+09,8.999999E+09,8.999999E+09,8.999999E+09,8.999999E+09,8.999999E+09]];
	LOCAL CONST Robtarget Tr_meulage_bavure_P5 :=[[-26.540828125,-187.172171875,120.8461796875],[0.669531680140477,-0.714893539407899,0.147166336255855,-0.137828248462155],[0,0,0,0],[8.999999E+09,8.999999E+09,8.999999E+09,8.999999E+09,8.999999E+09,8.999999E+09]];
	LOCAL CONST Robtarget Tr_meulage_bavure_P6 :=[[-30.04144921875,-185.659375,120.70628125],[0.669679719549337,-0.714756413562282,0.147133931327499,-0.137854810391296],[0,0,0,0],[8.999999E+09,8.999999E+09,8.999999E+09,8.999999E+09,8.999999E+09,8.999999E+09]];
	LOCAL CONST Robtarget Tr_meulage_bavure_P7 :=[[-30.068529296875,-185.646375,120.705],[0.669870848233334,-0.714597401624903,0.147046984367024,-0.137843333776627],[0,0,0,0],[8.999999E+09,8.999999E+09,8.999999E+09,8.999999E+09,8.999999E+09,8.999999E+09]];
	LOCAL CONST Robtarget Tr_meulage_bavure_P8 :=[[-30.0791953125,-185.641921875,120.70459375],[0.670099032585084,-0.714426214555078,0.146896426058777,-0.137782112395602],[0,0,0,0],[8.999999E+09,8.999999E+09,8.999999E+09,8.999999E+09,8.999999E+09,8.999999E+09]];
	LOCAL CONST Robtarget Tr_meulage_bavure_P9 :=[[-30.084818359375,-185.63915625,120.7043203125],[0.670361285794342,-0.714248666633679,0.146675136209692,-0.13766260617189],[0,0,0,0],[8.999999E+09,8.999999E+09,8.999999E+09,8.999999E+09,8.999999E+09,8.999999E+09]];
	LOCAL CONST Robtarget Tr_meulage_bavure_P10 :=[[-30.094623046875,-185.636203125,120.704125],[0.670663360246388,-0.71405968398396,0.146380908619124,-0.137484742875675],[0,0,0,0],[8.999999E+09,8.999999E+09,8.999999E+09,8.999999E+09,8.999999E+09,8.999999E+09]];
	LOCAL CONST Robtarget Tr_meulage_bavure_P11 :=[[-30.142390625,-185.6151875,120.70215625],[0.671007992547219,-0.713853828420596,0.146019976696523,-0.137255790378974],[0,0,0,0],[8.999999E+09,8.999999E+09,8.999999E+09,8.999999E+09,8.999999E+09,8.999999E+09]];
	LOCAL CONST Robtarget Tr_meulage_bavure_P12 :=[[-35.70280078125,-183.208296875,120.479328125],[0.671385782307399,-0.71363421910184,0.145608002278452,-0.136987745126591],[0,0,0,0],[8.999999E+09,8.999999E+09,8.999999E+09,8.999999E+09,8.999999E+09,8.999999E+09]];
	LOCAL CONST Robtarget Tr_meulage_bavure_P13 :=[[-38.21288671875,-182.114109375,120.3775703125],[0.67178864416036,-0.71340025939979,0.145166715828395,-0.136699349234353],[0,0,0,0],[8.999999E+09,8.999999E+09,8.999999E+09,8.999999E+09,8.999999E+09,8.999999E+09]];
	LOCAL CONST Robtarget Tr_meulage_bavure_P14 :=[[-40.73563671875,-181.00378125,120.2736640625],[0.672219125947048,-0.713138793119268,0.144722380186128,-0.136418258061899],[0,0,0,0],[8.999999E+09,8.999999E+09,8.999999E+09,8.999999E+09,8.999999E+09,8.999999E+09]];
	LOCAL CONST Robtarget Tr_meulage_bavure_P15 :=[[-45.13174609375,-179.22815625,120.1169765625],[0.672659005353849,-0.712855439880195,0.144307461643643,-0.136170264241325],[0,0,0,0],[8.999999E+09,8.999999E+09,8.999999E+09,8.999999E+09,8.999999E+09,8.999999E+09]];
	LOCAL CONST Robtarget Tr_meulage_bavure_P16 :=[[-48.7796875,-177.715328125,119.9809296875],[0.673112531326729,-0.712537142413095,0.143944029666039,-0.13597962044441],[0,0,0,0],[8.999999E+09,8.999999E+09,8.999999E+09,8.999999E+09,8.999999E+09,8.999999E+09]];
	LOCAL CONST Robtarget Tr_meulage_bavure_P17 :=[[-50.484296875,-176.978171875,119.9127265625],[0.673572342368902,-0.712181734825259,0.143656580981382,-0.135868550142021],[0,0,0,0],[8.999999E+09,8.999999E+09,8.999999E+09,8.999999E+09,8.999999E+09,8.999999E+09]];
	LOCAL CONST Robtarget Tr_meulage_bavure_P18 :=[[-52.23214453125,-176.16971875,119.8347421875],[0.674040154897297,-0.711785020012287,0.143451311140535,-0.135844308692697],[0,0,0,0],[8.999999E+09,8.999999E+09,8.999999E+09,8.999999E+09,8.999999E+09,8.999999E+09]];
	LOCAL CONST Robtarget Tr_meulage_bavure_P19 :=[[-54.175390625,-175.414875,119.7700859375],[0.674508593884136,-0.711356366129925,0.143323487961932,-0.135899429510575],[0,0,0,0],[8.999999E+09,8.999999E+09,8.999999E+09,8.999999E+09,8.999999E+09,8.999999E+09]];
	LOCAL CONST Robtarget Tr_meulage_bavure_P20 :=[[-57.50351171875,-173.996859375,119.640171875],[0.674979414736806,-0.710894404940432,0.143271780368882,-0.136033568121544],[0,0,0,0],[8.999999E+09,8.999999E+09,8.999999E+09,8.999999E+09,8.999999E+09,8.999999E+09]];
	LOCAL CONST Robtarget Tr_meulage_bavure_P21 :=[[-60.803421875,-172.5603125,119.5066796875],[0.675453329128334,-0.710399765132998,0.143292361576134,-0.136243432804543],[0,0,0,0],[8.999999E+09,8.999999E+09,8.999999E+09,8.999999E+09,8.999999E+09,8.999999E+09]];
	LOCAL CONST Robtarget Tr_meulage_bavure_P22 :=[[-66.3370234375,-170.2145,119.2925],[0.675935334208242,-0.709875638276012,0.143363839988407,-0.136509382588874],[0,0,0,0],[8.999999E+09,8.999999E+09,8.999999E+09,8.999999E+09,8.999999E+09,8.999999E+09]];
	LOCAL CONST Robtarget Tr_meulage_bavure_P23 :=[[-68.5413984375,-169.262671875,119.2045234375],[0.676419098857861,-0.709329836224235,0.143482466854611,-0.136825318737922],[0,0,0,0],[8.999999E+09,8.999999E+09,8.999999E+09,8.999999E+09,8.999999E+09,8.999999E+09]];
	LOCAL CONST Robtarget Tr_meulage_bavure_P24 :=[[-69.8784453125,-168.719875,119.156453125],[0.676900877136821,-0.708747902067837,0.143693258530057,-0.137236515909057],[0,0,0,0],[8.999999E+09,8.999999E+09,8.999999E+09,8.999999E+09,8.999999E+09,8.999999E+09]];
	LOCAL CONST Robtarget Tr_meulage_bavure_P25 :=[[-70.8627109375,-168.2819375,119.1151875],[0.677364190551129,-0.708114541202655,0.144075036563725,-0.137818481110222],[0,0,0,0],[8.999999E+09,8.999999E+09,8.999999E+09,8.999999E+09,8.999999E+09,8.999999E+09]];
	LOCAL CONST Robtarget Tr_meulage_bavure_P26 :=[[-73.6882578125,-167.151109375,119.016078125],[0.677775243324627,-0.707407630411471,0.144765533581592,-0.138701493354279],[0,0,0,0],[8.999999E+09,8.999999E+09,8.999999E+09,8.999999E+09,8.999999E+09,8.999999E+09]];
	LOCAL CONST Robtarget Tr_meulage_bavure_P27 :=[[-76.772765625,-165.861484375,118.8994375],[0.678091352221753,-0.706582066090861,0.145975480315782,-0.140089475220023],[0,0,0,0],[8.999999E+09,8.999999E+09,8.999999E+09,8.999999E+09,8.999999E+09,8.999999E+09]];
	LOCAL CONST Robtarget Tr_meulage_bavure_P28 :=[[-78.1794140625,-165.266765625,118.8452421875],[0.678253171150839,-0.70556182147809,0.148017415956871,-0.142288427041001],[0,0,0,0],[8.999999E+09,8.999999E+09,8.999999E+09,8.999999E+09,8.999999E+09,8.999999E+09]];
	LOCAL CONST Robtarget Tr_meulage_bavure_P29 :=[[-80.7164921875,-164.21375,118.750484375],[0.678150988954776,-0.704262766580497,0.151313446508017,-0.145703235015249],[0,0,0,0],[8.999999E+09,8.999999E+09,8.999999E+09,8.999999E+09,8.999999E+09,8.999999E+09]];
	LOCAL CONST Robtarget Tr_meulage_bavure_P30 :=[[-83.2541796875,-163.142453125,118.6529453125],[0.677652656901611,-0.702539417257042,0.156409338563409,-0.150868693255027],[0,0,0,0],[8.999999E+09,8.999999E+09,8.999999E+09,8.999999E+09,8.999999E+09,8.999999E+09]];
	LOCAL CONST Robtarget Tr_meulage_bavure_P31 :=[[-89.7933359375,-160.3963125,118.4038203125],[0.676559483874496,-0.700182932364687,0.164005354809088,-0.158471983639409],[0,0,0,0],[8.999999E+09,8.999999E+09,8.999999E+09,8.999999E+09,8.999999E+09,8.999999E+09]];
	LOCAL CONST Robtarget Tr_meulage_bavure_P32 :=[[-99.22696875,-156.344125,118.0305625],[0.674577470384258,-0.696900432513931,0.174934418013698,-0.169330957022277],[0,0,0,0],[8.999999E+09,8.999999E+09,8.999999E+09,8.999999E+09,8.999999E+09,8.999999E+09]];
	LOCAL CONST Robtarget Tr_meulage_bavure_P33 :=[[-99.479734375,-156.240140625,118.021265625],[0.671257622414274,-0.692247177276975,0.190220987212299,-0.184453316388656],[0,0,0,0],[8.999999E+09,8.999999E+09,8.999999E+09,8.999999E+09,8.999999E+09,8.999999E+09]];
	LOCAL CONST Robtarget Tr_meulage_bavure_P34 :=[[-99.5415234375,-156.214390625,118.0189453125],[0.66593508245143,-0.685546501923063,0.211030781372233,-0.204993826675057],[0,0,0,0],[8.999999E+09,8.999999E+09,8.999999E+09,8.999999E+09,8.999999E+09,8.999999E+09]];
	LOCAL CONST Robtarget Tr_meulage_bavure_P35 :=[[-99.655125,-156.170546875,118.015203125],[0.657662452479807,-0.675817859748452,0.238501051782266,-0.232093876140712],[0,0,0,0],[8.999999E+09,8.999999E+09,8.999999E+09,8.999999E+09,8.999999E+09,8.999999E+09]];
	LOCAL CONST Robtarget Tr_meulage_bavure_P36 :=[[-104.5490078125,-154.36715625,117.8673046875],[0.645148897160641,-0.6617739420746,0.273448251468535,-0.266578701047652],[0,0,0,0],[8.999999E+09,8.999999E+09,8.999999E+09,8.999999E+09,8.999999E+09,8.999999E+09]];
	LOCAL CONST Robtarget Tr_meulage_bavure_P37 :=[[-104.5672578125,-154.357375,117.8662890625],[0.626979244435916,-0.641982178455581,0.315721764490947,-0.308343440044892],[0,0,0,0],[8.999999E+09,8.999999E+09,8.999999E+09,8.999999E+09,8.999999E+09,8.999999E+09]];
	LOCAL CONST Robtarget Tr_meulage_bavure_P38 :=[[-104.6088046875,-154.33671875,117.8642109375],[0.602238050245919,-0.615552776696801,0.363355171732101,-0.355495610538847],[0,0,0,0],[8.999999E+09,8.999999E+09,8.999999E+09,8.999999E+09,8.999999E+09,8.999999E+09]];
	LOCAL CONST Robtarget Tr_meulage_bavure_P39 :=[[-108.101734375,-151.681875,117.5492890625],[0.571545330590734,-0.58313852561273,0.412296731017639,-0.404099988391869],[0,0,0,0],[8.999999E+09,8.999999E+09,8.999999E+09,8.999999E+09,8.999999E+09,8.999999E+09]];
	LOCAL CONST Robtarget Tr_meulage_bavure_P40 :=[[-109.2002109375,-149.8225,117.2934296875],[0.537536586461242,-0.54746985134436,0.457636343759209,-0.449333013426882],[0,0,0,0],[8.999999E+09,8.999999E+09,8.999999E+09,8.999999E+09,8.999999E+09,8.999999E+09]];
	LOCAL CONST Robtarget Tr_meulage_bavure_P41 :=[[-109.2302578125,-149.46471875,117.239453125],[0.503963303805163,-0.512367230000639,0.495729913433932,-0.487598875066425],[0,0,0,0],[8.999999E+09,8.999999E+09,8.999999E+09,8.999999E+09,8.999999E+09,8.999999E+09]];
	LOCAL CONST Robtarget Tr_meulage_bavure_P42 :=[[-108.914109375,-148.094828125,117.0214765625],[0.473967645524778,-0.481029150504827,0.525361611619012,-0.517649306381624],[0,0,0,0],[8.999999E+09,8.999999E+09,8.999999E+09,8.999999E+09,8.999999E+09,8.999999E+09]];
	LOCAL CONST Robtarget Tr_meulage_bavure_P43 :=[[-108.7151875,-146.81065625,116.8196953125],[0.44916760927619,-0.455064944042426,0.547208865012099,-0.540117407174539],[0,0,0,0],[8.999999E+09,8.999999E+09,8.999999E+09,8.999999E+09,8.999999E+09,8.999999E+09]];
	LOCAL CONST Robtarget Tr_meulage_bavure_P44 :=[[-108.6124140625,-146.52896875,116.7738828125],[0.42979227134837,-0.434687863037518,0.562769337460544,-0.556431251846358],[0,0,0,0],[8.999999E+09,8.999999E+09,8.999999E+09,8.999999E+09,8.999999E+09,8.999999E+09]];
	LOCAL CONST Robtarget Tr_meulage_bavure_P45 :=[[-107.3795390625,-144.0755625,116.366046875],[0.415317742201116,-0.419327569666871,0.573557763210722,-0.568073106730952],[0,0,0,0],[8.999999E+09,8.999999E+09,8.999999E+09,8.999999E+09,8.999999E+09,8.999999E+09]];
	LOCAL CONST Robtarget Tr_meulage_bavure_P46 :=[[-106.6686953125,-142.77896875,116.1489609375],[0.404919768534327,-0.408143315102881,0.580847369204519,-0.576259793040541],[0,0,0,0],[8.999999E+09,8.999999E+09,8.999999E+09,8.999999E+09,8.999999E+09,8.999999E+09]];
	LOCAL CONST Robtarget Tr_meulage_bavure_P47 :=[[-105.4624375,-140.42771875,115.757453125],[0.397727870790555,-0.400228968360671,0.585620285765671,-0.581960646935082],[0,0,0,0],[8.999999E+09,8.999999E+09,8.999999E+09,8.999999E+09,8.999999E+09,8.999999E+09]];
	LOCAL CONST Robtarget Tr_meulage_bavure_P48 :=[[-104.91825,-139.05621875,115.533265625],[0.392946478014115,-0.394770373643393,0.588618518253814,-0.585899016451166],[0,0,0,0],[8.999999E+09,8.999999E+09,8.999999E+09,8.999999E+09,8.999999E+09,8.999999E+09]];
	LOCAL CONST Robtarget Tr_meulage_bavure_P49 :=[[-101.483453125,-131.47175,114.2823359375],[0.389911509100262,-0.39108620095069,0.590386035835644,-0.588612714089142],[0,0,0,0],[8.999999E+09,8.999999E+09,8.999999E+09,8.999999E+09,8.999999E+09,8.999999E+09]];
	LOCAL CONST Robtarget Tr_meulage_bavure_P50 :=[[-101.1290625,-130.6462265625,114.1466953125],[0.388052766691468,-0.388599096660154,0.591349460369008,-0.590518084447286],[0,0,0,0],[8.999999E+09,8.999999E+09,8.999999E+09,8.999999E+09,8.999999E+09,8.999999E+09]];
	LOCAL CONST Robtarget Tr_meulage_bavure_P51 :=[[-99.405671875,-126.421421875,113.454859375],[0.386942192177987,-0.386879904880759,0.591813692097883,-0.591908973540207],[0,0,0,0],[8.999999E+09,8.999999E+09,8.999999E+09,8.999999E+09,8.999999E+09,8.999999E+09]];
	LOCAL CONST Robtarget Tr_meulage_bavure_P52 :=[[-97.58875,-122.258453125,112.7700390625],[0.386234783892369,-0.385576961066301,0.592011906779583,-0.593021922898043],[0,0,0,0],[8.999999E+09,8.999999E+09,8.999999E+09,8.999999E+09,8.999999E+09,8.999999E+09]];
	LOCAL CONST Robtarget Tr_meulage_bavure_P53 :=[[-96.83659375,-120.6601875,112.5056875],[0.385658080196084,-0.384416144697278,0.592124551178156,-0.594037531446978],[0,0,0,0],[8.999999E+09,8.999999E+09,8.999999E+09,8.999999E+09,8.999999E+09,8.999999E+09]];
	LOCAL CONST Robtarget Tr_meulage_bavure_P54 :=[[-95.875421875,-118.5384375,112.155734375],[0.385012820824944,-0.383198311915761,0.59228124607711,-0.595085798091903],[0,0,0,0],[8.999999E+09,8.999999E+09,8.999999E+09,8.999999E+09,8.999999E+09,8.999999E+09]];
	LOCAL CONST Robtarget Tr_meulage_bavure_P55 :=[[-94.98903125,-116.536390625,111.8260625],[0.384130202280648,-0.381750830880857,0.592587227017346,-0.596280696646719],[0,0,0,0],[8.999999E+09,8.999999E+09,8.999999E+09,8.999999E+09,8.999999E+09,8.999999E+09]];
	LOCAL CONST Robtarget Tr_meulage_bavure_P56 :=[[-93.545078125,-113.0680390625,111.2573359375],[0.38288932018167,-0.379963921653615,0.593121119963392,-0.597687647342486],[0,0,0,0],[8.999999E+09,8.999999E+09,8.999999E+09,8.999999E+09,8.999999E+09,8.999999E+09]];
	LOCAL CONST Robtarget Tr_meulage_bavure_P57 :=[[-91.181328125,-107.8744921875,110.4004453125],[0.381206757803961,-0.377751579452106,0.59392870913424,-0.599361193682213],[0,0,0,0],[8.999999E+09,8.999999E+09,8.999999E+09,8.999999E+09,8.999999E+09,8.999999E+09]];
	LOCAL CONST Robtarget Tr_meulage_bavure_P58 :=[[-89.0887109375,-103.1712890625,109.6257109375],[0.379070079610735,-0.375106095178924,0.595012198926034,-0.601300070873717],[0,0,0,0],[8.999999E+09,8.999999E+09,8.999999E+09,8.999999E+09,8.999999E+09,8.999999E+09]];
	LOCAL CONST Robtarget Tr_meulage_bavure_P59 :=[[-87.8623984375,-100.3644765625,109.1639453125],[0.376548072931825,-0.372095884855012,0.596320265887,-0.603455335329594],[0,0,0,0],[8.999999E+09,8.999999E+09,8.999999E+09,8.999999E+09,8.999999E+09,8.999999E+09]];
	LOCAL CONST Robtarget Tr_meulage_bavure_P60 :=[[-84.9622578125,-93.4823515625,108.03453125],[0.373781897414602,-0.368854705244238,0.597755610637525,-0.605740480350857],[0,0,0,0],[8.999999E+09,8.999999E+09,8.999999E+09,8.999999E+09,8.999999E+09,8.999999E+09]];
	LOCAL CONST Robtarget Tr_meulage_bavure_P61 :=[[-84.9034375,-93.3372109375,108.0107734375],[0.3709848576004,-0.365598343256536,0.599187285812621,-0.608015364410959],[0,0,0,0],[8.999999E+09,8.999999E+09,8.999999E+09,8.999999E+09,8.999999E+09,8.999999E+09]];
	LOCAL CONST Robtarget Tr_meulage_bavure_P62 :=[[-82.5685703125,-88.3507578125,107.1863359375],[0.368435774896412,-0.362598150549834,0.600447878483731,-0.610114748402877],[0,0,0,0],[8.999999E+09,8.999999E+09,8.999999E+09,8.999999E+09,8.999999E+09,8.999999E+09]];
	LOCAL CONST Robtarget Tr_meulage_bavure_P63 :=[[-82.4626015625,-88.1271015625,107.1493203125],[0.366428540766891,-0.360141466039184,0.601369839268845,-0.61186809474621],[0,0,0,0],[8.999999E+09,8.999999E+09,8.999999E+09,8.999999E+09,8.999999E+09,8.999999E+09]];
	LOCAL CONST Robtarget Tr_meulage_bavure_P64 :=[[-82.364390625,-87.846921875,107.103859375],[0.36523794914622,-0.358496702526157,0.601802620814896,-0.613119042569758],[0,0,0,0],[8.999999E+09,8.999999E+09,8.999999E+09,8.999999E+09,8.999999E+09,8.999999E+09]];
	LOCAL CONST Robtarget Tr_meulage_bavure_P65 :=[[-81.0823203125,-84.5063203125,106.5589296875],[0.365059720589847,-0.357854316583918,0.601642844610744,-0.613756935629905],[0,0,0,0],[8.999999E+09,8.999999E+09,8.999999E+09,8.999999E+09,8.999999E+09,8.999999E+09]];
	LOCAL CONST Robtarget Tr_meulage_bavure_P66 :=[[-80.90546875,-84.3459375,106.52975],[0.365956742000585,-0.358263127593111,0.600853906612777,-0.613757099592081],[0,0,0,0],[8.999999E+09,8.999999E+09,8.999999E+09,8.999999E+09,8.999999E+09,8.999999E+09]];
	LOCAL CONST Robtarget Tr_meulage_bavure_P67 :=[[-76.770609375,-74.70728125,104.946046875],[0.367866745064765,-0.359661152903732,0.599471899012635,-0.61314872197665],[0,0,0,0],[8.999999E+09,8.999999E+09,8.999999E+09,8.999999E+09,8.999999E+09,8.999999E+09]];
	LOCAL CONST Robtarget Tr_meulage_bavure_P68 :=[[-76.7337109375,-74.6066875,104.9296796875],[0.370588353593622,-0.361851510179718,0.597609212634273,-0.612038385835456],[0,0,0,0],[8.999999E+09,8.999999E+09,8.999999E+09,8.999999E+09,8.999999E+09,8.999999E+09]];
	LOCAL CONST Robtarget Tr_meulage_bavure_P69 :=[[-76.650359375,-74.46253125,104.9054375],[0.373843491928935,-0.364549884334191,0.595415082095045,-0.610594223185954],[0,0,0,0],[8.999999E+09,8.999999E+09,8.999999E+09,8.999999E+09,8.999999E+09,8.999999E+09]];
	LOCAL CONST Robtarget Tr_meulage_bavure_P70 :=[[-76.62025,-74.3851328125,104.892796875],[0.377319950232188,-0.367455112532482,0.593071388272393,-0.608993205087853],[0,0,0,0],[8.999999E+09,8.999999E+09,8.999999E+09,8.999999E+09,8.999999E+09,8.999999E+09]];
	LOCAL CONST Robtarget Tr_meulage_bavure_P71 :=[[-76.387890625,-73.865828125,104.80721875],[0.380721235594171,-0.370276875671202,0.590754110860475,-0.607417448393006],[0,0,0,0],[8.999999E+09,8.999999E+09,8.999999E+09,8.999999E+09,8.999999E+09,8.999999E+09]];
	LOCAL CONST Robtarget Tr_meulage_bavure_P72 :=[[-76.3263515625,-73.7296875,104.7847734375],[0.383800799794269,-0.372777948903862,0.588617325218217,-0.606022434684774],[0,0,0,0],[8.999999E+09,8.999999E+09,8.999999E+09,8.999999E+09,8.999999E+09,8.999999E+09]];
	LOCAL CONST Robtarget Tr_meulage_bavure_P73 :=[[-74.7453046875,-70.30503125,104.219140625],[0.386394391843568,-0.374787876001239,0.586761945802403,-0.604932922655476],[0,0,0,0],[8.999999E+09,8.999999E+09,8.999999E+09,8.999999E+09,8.999999E+09,8.999999E+09]];
	LOCAL CONST Robtarget Tr_meulage_bavure_P74 :=[[-74.4052734375,-69.4974765625,104.086625],[0.388419708333068,-0.376243160995329,0.585252977577213,-0.604193815112091],[0,0,0,0],[8.999999E+09,8.999999E+09,8.999999E+09,8.999999E+09,8.999999E+09,8.999999E+09]];
	LOCAL CONST Robtarget Tr_meulage_bavure_P75 :=[[-73.7152421875,-67.988265625,103.83753125],[0.389889511546769,-0.37714076028119,0.584079201862099,-0.603823237108743],[0,0,0,0],[8.999999E+09,8.999999E+09,8.999999E+09,8.999999E+09,8.999999E+09,8.999999E+09]];
	LOCAL CONST Robtarget Tr_meulage_bavure_P76 :=[[-71.55009375,-62.897828125,103.001625],[0.390860870731665,-0.377555153366475,0.583216532347255,-0.603770123717749],[0,0,0,0],[8.999999E+09,8.999999E+09,8.999999E+09,8.999999E+09,8.999999E+09,8.999999E+09]];
	LOCAL CONST Robtarget Tr_meulage_bavure_P77 :=[[-69.3719765625,-57.6667265625,102.14384375],[0.39144189175867,-0.377573402482734,0.582589135930907,-0.603987971576657],[0,0,0,0],[8.999999E+09,8.999999E+09,8.999999E+09,8.999999E+09,8.999999E+09,8.999999E+09]];
	LOCAL CONST Robtarget Tr_meulage_bavure_P78 :=[[-68.8868359375,-56.3606953125,101.93121875],[0.391764626474994,-0.377335763884371,0.582119936863275,-0.604379498198775],[0,0,0,0],[8.999999E+09,8.999999E+09,8.999999E+09,8.999999E+09,8.999999E+09,8.999999E+09]];
	LOCAL CONST Robtarget Tr_meulage_bavure_P79 :=[[-68.004375,-54.4609375,101.6173046875],[0.391964682468506,-0.376966917039535,0.581720448343724,-0.604864407230122],[0,0,0,0],[8.999999E+09,8.999999E+09,8.999999E+09,8.999999E+09,8.999999E+09,8.999999E+09]];
	LOCAL CONST Robtarget Tr_meulage_bavure_P80 :=[[-66.567140625,-51.3191328125,101.0987421875],[0.392172056625141,-0.37659362621559,0.581310026590637,-0.605356896121117],[0,0,0,0],[8.999999E+09,8.999999E+09,8.999999E+09,8.999999E+09,8.999999E+09,8.999999E+09]];
	LOCAL CONST Robtarget Tr_meulage_bavure_P81 :=[[-63.55097265625,-44.5826328125,99.988578125],[0.39250282655565,-0.37632875199332,0.580817322810993,-0.605780025332337],[0,0,0,0],[8.999999E+09,8.999999E+09,8.999999E+09,8.999999E+09,8.999999E+09,8.999999E+09]];
	LOCAL CONST Robtarget Tr_meulage_bavure_P82 :=[[-61.5196328125,-40.20978125,99.266015625],[0.393036143496634,-0.376245415313896,0.580192446573228,-0.606084731947554],[0,0,0,0],[8.999999E+09,8.999999E+09,8.999999E+09,8.999999E+09,8.999999E+09,8.999999E+09]];
	LOCAL CONST Robtarget Tr_meulage_bavure_P83 :=[[-61.34173046875,-39.7959296875,99.1980078125],[0.393844037957916,-0.376409284270551,0.579389809423971,-0.606226338272753],[0,0,0,0],[8.999999E+09,8.999999E+09,8.999999E+09,8.999999E+09,8.999999E+09,8.999999E+09]];
	LOCAL CONST Robtarget Tr_meulage_bavure_P84 :=[[-59.2306484375,-35.2144609375,98.4414296875],[0.394945191901318,-0.376841298690639,0.578399869593115,-0.606186870403716],[0,0,0,0],[8.999999E+09,8.999999E+09,8.999999E+09,8.999999E+09,8.999999E+09,8.999999E+09]];
	LOCAL CONST Robtarget Tr_meulage_bavure_P85 :=[[-58.6750625,-33.9638515625,98.2354453125],[0.396322909058589,-0.377519574437418,0.577230153395589,-0.605980587711218],[0,0,0,0],[8.999999E+09,8.999999E+09,8.999999E+09,8.999999E+09,8.999999E+09,8.999999E+09]];
	LOCAL CONST Robtarget Tr_meulage_bavure_P86 :=[[-56.72388671875,-29.005845703125,97.42540625],[0.39792478852545,-0.378391130330531,0.575911518316492,-0.605641757340553],[0,0,0,0],[8.999999E+09,8.999999E+09,8.999999E+09,8.999999E+09,8.999999E+09,8.999999E+09]];
	LOCAL CONST Robtarget Tr_meulage_bavure_P87 :=[[-56.24359765625,-27.959251953125,97.252625],[0.399660043677932,-0.379375131484399,0.574502955356672,-0.605221210290087],[0,0,0,0],[8.999999E+09,8.999999E+09,8.999999E+09,8.999999E+09,8.999999E+09,8.999999E+09]];
	LOCAL CONST Robtarget Tr_meulage_bavure_P88 :=[[-55.6716015625,-26.676513671875,97.0412890625],[0.401432845225554,-0.380375288828059,0.573061720506622,-0.604786387837124],[0,0,0,0],[8.999999E+09,8.999999E+09,8.999999E+09,8.999999E+09,8.999999E+09,8.999999E+09]];
	LOCAL CONST Robtarget Tr_meulage_bavure_P89 :=[[-53.16237109375,-21.358171875,96.161484375],[0.40313595732091,-0.38128615844512,0.571653580760205,-0.604412482413419],[0,0,0,0],[8.999999E+09,8.999999E+09,8.999999E+09,8.999999E+09,8.999999E+09,8.999999E+09]];
	LOCAL CONST Robtarget Tr_meulage_bavure_P90 :=[[-52.82059375,-20.613361328125,96.0385234375],[0.404658938274494,-0.382008498988228,0.570351167311481,-0.60416901304333],[0,0,0,0],[8.999999E+09,8.999999E+09,8.999999E+09,8.999999E+09,8.999999E+09,8.999999E+09]];
	LOCAL CONST Robtarget Tr_meulage_bavure_P91 :=[[-52.7305,-20.431427734375,96.0083125],[0.405909529628385,-0.382458956577102,0.56921502241095,-0.60411659350867],[0,0,0,0],[8.999999E+09,8.999999E+09,8.999999E+09,8.999999E+09,8.999999E+09,8.999999E+09]];
	LOCAL CONST Robtarget Tr_meulage_bavure_P92 :=[[-52.49386328125,-19.87358984375,95.9167265625],[0.406822753257539,-0.382574612079536,0.568285439359878,-0.604304205707439],[0,0,0,0],[8.999999E+09,8.999999E+09,8.999999E+09,8.999999E+09,8.999999E+09,8.999999E+09]];
	LOCAL CONST Robtarget Tr_meulage_bavure_P93 :=[[-50.4593671875,-14.2934619140625,95.00928125],[0.407361701610647,-0.382326138018453,0.567587387642003,-0.60475426880552],[0,0,0,0],[8.999999E+09,8.999999E+09,8.999999E+09,8.999999E+09,8.999999E+09,8.999999E+09]];
	LOCAL CONST Robtarget Tr_meulage_bavure_P94 :=[[-49.81048046875,-12.78501953125,94.761390625],[0.40752717216672,-0.381713045724037,0.56711774569736,-0.605470244673528],[0,0,0,0],[8.999999E+09,8.999999E+09,8.999999E+09,8.999999E+09,8.999999E+09,8.999999E+09]];
	LOCAL CONST Robtarget Tr_meulage_bavure_P95 :=[[-47.11734375,-6.72971044921875,93.763953125],[0.407346055552551,-0.380768592319307,0.566860430220131,-0.606427013563545],[0,0,0,0],[8.999999E+09,8.999999E+09,8.999999E+09,8.999999E+09,8.999999E+09,8.999999E+09]];
	LOCAL CONST Robtarget Tr_meulage_bavure_P96 :=[[-46.71208203125,-5.6802802734375,93.592703125],[0.406879226873067,-0.379549274784459,0.566773571736086,-0.607584859201812],[0,0,0,0],[8.999999E+09,8.999999E+09,8.999999E+09,8.999999E+09,8.999999E+09,8.999999E+09]];
	LOCAL CONST Robtarget Tr_meulage_bavure_P97 :=[[-43.66248046875,1.60443225097656,92.3977421875],[0.40620948211355,-0.37813276478203,0.56680235526825,-0.60888796908931],[0,0,0,0],[8.999999E+09,8.999999E+09,8.999999E+09,8.999999E+09,8.999999E+09,8.999999E+09]];
	LOCAL CONST Robtarget Tr_meulage_bavure_P98 :=[[-43.61665625,1.70914001464844,92.380515625],[0.405424359221477,-0.376606001289049,0.566892586617245,-0.610271909874064],[0,0,0,0],[8.999999E+09,8.999999E+09,8.999999E+09,8.999999E+09,8.999999E+09,8.999999E+09]];
	LOCAL CONST Robtarget Tr_meulage_bavure_P99 :=[[-43.487640625,2.03753186035156,92.3268671875],[0.404622741462155,-0.375067557992027,0.566985365152845,-0.61166360013985],[0,0,0,0],[8.999999E+09,8.999999E+09,8.999999E+09,8.999999E+09,8.999999E+09,8.999999E+09]];
	LOCAL CONST Robtarget Tr_meulage_bavure_P100 :=[[-40.9436171875,8.11401806640625,91.3301015625],[0.403904652027587,-0.37359638742574,0.567012562464698,-0.613011847667014],[0,0,0,0],[8.999999E+09,8.999999E+09,8.999999E+09,8.999999E+09,8.999999E+09,8.999999E+09]];
	LOCAL CONST Robtarget Tr_meulage_bavure_P101 :=[[-39.297953125,11.4520546875,90.7760390625],[0.403328174823348,-0.372263494520579,0.56694899381121,-0.61425980859686],[0,0,0,0],[8.999999E+09,8.999999E+09,8.999999E+09,8.999999E+09,8.999999E+09,8.999999E+09]];
	LOCAL CONST Robtarget Tr_meulage_bavure_P102 :=[[-38.01172265625,14.0978330078125,90.337359375],[0.402952069393615,-0.371111755406661,0.566755310169034,-0.615381274630283],[0,0,0,0],[8.999999E+09,8.999999E+09,8.999999E+09,8.999999E+09,8.999999E+09,8.999999E+09]];
	LOCAL CONST Robtarget Tr_meulage_bavure_P103 :=[[-37.25991796875,15.4117021484375,90.1165546875],[0.402772976850783,-0.370148033385059,0.566441146031082,-0.616367415250779],[0,0,0,0],[8.999999E+09,8.999999E+09,8.999999E+09,8.999999E+09,8.999999E+09,8.999999E+09]];
	LOCAL CONST Robtarget Tr_meulage_bavure_P104 :=[[-36.9197890625,16.2553974609375,89.9785],[0.40277574572886,-0.369352578779167,0.566014636258763,-0.617233993508621],[0,0,0,0],[8.999999E+09,8.999999E+09,8.999999E+09,8.999999E+09,8.999999E+09,8.999999E+09]];
	LOCAL CONST Robtarget Tr_meulage_bavure_P105 :=[[-35.35371484375,20.598912109375,89.272609375],[0.402919244920223,-0.36868653017654,0.565501410726196,-0.618008478102026],[0,0,0,0],[8.999999E+09,8.999999E+09,8.999999E+09,8.999999E+09,8.999999E+09,8.999999E+09]];
	LOCAL CONST Robtarget Tr_meulage_bavure_P106 :=[[-35.23979296875,20.8933671875,89.2245546875],[0.403104648947737,-0.368064859173333,0.564964303779566,-0.618748928801745],[0,0,0,0],[8.999999E+09,8.999999E+09,8.999999E+09,8.999999E+09,8.999999E+09,8.999999E+09]];
	LOCAL CONST Robtarget Tr_meulage_bavure_P107 :=[[-34.034171875,23.65528515625,88.7702109375],[0.403246861560216,-0.367415908699814,0.564457395124475,-0.619504130547504],[0,0,0,0],[8.999999E+09,8.999999E+09,8.999999E+09,8.999999E+09,8.999999E+09,8.999999E+09]];
	LOCAL CONST Robtarget Tr_meulage_bavure_P108 :=[[-31.766767578125,28.729400390625,87.9341171875],[0.403250236486079,-0.366650971562574,0.56403602497994,-0.620338354731489],[0,0,0,0],[8.999999E+09,8.999999E+09,8.999999E+09,8.999999E+09,8.999999E+09,8.999999E+09]];
	LOCAL CONST Robtarget Tr_meulage_bavure_P109 :=[[-30.2750546875,31.87352734375,87.4137734375],[0.403011674581128,-0.365672932276652,0.563757746101228,-0.621322863302465],[0,0,0,0],[8.999999E+09,8.999999E+09,8.999999E+09,8.999999E+09,8.999999E+09,8.999999E+09]];
	LOCAL CONST Robtarget Tr_meulage_bavure_P110 :=[[-27.227234375,38.65832421875,86.295390625],[0.402420856012029,-0.364390335566612,0.563689363657402,-0.622520232034036],[0,0,0,0],[8.999999E+09,8.999999E+09,8.999999E+09,8.999999E+09,8.999999E+09,8.999999E+09]];
	LOCAL CONST Robtarget Tr_meulage_bavure_P111 :=[[-25.943298828125,41.5028984375,85.8263359375],[0.401328624547936,-0.362670939389861,0.56391480998587,-0.624023406547493],[0,0,0,0],[8.999999E+09,8.999999E+09,8.999999E+09,8.999999E+09,8.999999E+09,8.999999E+09]];
	LOCAL CONST Robtarget Tr_meulage_bavure_P112 :=[[-25.105419921875,43.6431171875,85.47678125],[0.39956506746556,-0.360366895137582,0.564527602650736,-0.625932938576932],[0,0,0,0],[8.999999E+09,8.999999E+09,8.999999E+09,8.999999E+09,8.999999E+09,8.999999E+09]];
	LOCAL CONST Robtarget Tr_meulage_bavure_P113 :=[[-24.2619140625,45.3304140625,85.1964140625],[0.396896380792921,-0.357269109715579,0.565649118865714,-0.628389306467703],[0,0,0,0],[8.999999E+09,8.999999E+09,8.999999E+09,8.999999E+09,8.999999E+09,8.999999E+09]];
	LOCAL CONST Robtarget Tr_meulage_bavure_P114 :=[[-21.813923828125,51.13175390625,84.24428125],[0.393016102257896,-0.353119341686348,0.567439841612525,-0.631551343948981],[0,0,0,0],[8.999999E+09,8.999999E+09,8.999999E+09,8.999999E+09,8.999999E+09,8.999999E+09]];
	LOCAL CONST Robtarget Tr_meulage_bavure_P115 :=[[-20.728291015625,53.338671875,83.87803125],[0.387548152467338,-0.347573184346433,0.570065323650296,-0.635629481548737],[0,0,0,0],[8.999999E+09,8.999999E+09,8.999999E+09,8.999999E+09,8.999999E+09,8.999999E+09]];
	LOCAL CONST Robtarget Tr_meulage_bavure_P116 :=[[-17.18916015625,61.0465234375,82.605484375],[0.379989704263492,-0.34019575019333,0.573742007357684,-0.640854730182525],[0,0,0,0],[8.999999E+09,8.999999E+09,8.999999E+09,8.999999E+09,8.999999E+09,8.999999E+09]];
	LOCAL CONST Robtarget Tr_meulage_bavure_P117 :=[[-16.84749609375,61.79646484375,82.481734375],[0.369807746271793,-0.330515992914933,0.57864505760346,-0.647434403268718],[0,0,0,0],[8.999999E+09,8.999999E+09,8.999999E+09,8.999999E+09,8.999999E+09,8.999999E+09]];
	LOCAL CONST Robtarget Tr_meulage_bavure_P118 :=[[-16.762546875,62.00539453125,82.44753125],[0.356424907300467,-0.318037680306614,0.584910700110494,-0.655509566869389],[0,0,0,0],[8.999999E+09,8.999999E+09,8.999999E+09,8.999999E+09,8.999999E+09,8.999999E+09]];
	LOCAL CONST Robtarget Tr_meulage_bavure_P119 :=[[-16.7153046875,62.1158359375,82.429390625],[0.33926970082892,-0.302259415741343,0.592570572159944,-0.6651281325468],[0,0,0,0],[8.999999E+09,8.999999E+09,8.999999E+09,8.999999E+09,8.999999E+09,8.999999E+09]];
	LOCAL CONST Robtarget Tr_meulage_bavure_P120 :=[[-14.5000693359375,67.7231171875,81.5130546875],[0.317912789183504,-0.282815842771056,0.601489801453402,-0.676133623109226],[0,0,0,0],[8.999999E+09,8.999999E+09,8.999999E+09,8.999999E+09,8.999999E+09,8.999999E+09]];
	LOCAL CONST Robtarget Tr_meulage_bavure_P121 :=[[-13.89879296875,68.71796875,81.3450234375],[0.292270894227027,-0.259638721665928,0.611283710906063,-0.688111679438976],[0,0,0,0],[8.999999E+09,8.999999E+09,8.999999E+09,8.999999E+09,8.999999E+09,8.999999E+09]];
	LOCAL CONST Robtarget Tr_meulage_bavure_P122 :=[[-12.8285546875,70.41190625,81.0576953125],[0.262803957734882,-0.233156311614193,0.621347502952184,-0.700356691071367],[0,0,0,0],[8.999999E+09,8.999999E+09,8.999999E+09,8.999999E+09,8.999999E+09,8.999999E+09]];
	LOCAL CONST Robtarget Tr_meulage_bavure_P123 :=[[-10.605658203125,72.24846875,80.718359375],[0.230734423197535,-0.204448855383546,0.630887535172692,-0.711999444836711],[0,0,0,0],[8.999999E+09,8.999999E+09,8.999999E+09,8.999999E+09,8.999999E+09,8.999999E+09]];
	LOCAL CONST Robtarget Tr_meulage_bavure_P124 :=[[-10.1763662109375,72.5388828125,80.6626640625],[0.198051266140744,-0.1752884592819,0.639162742324884,-0.722163860108188],[0,0,0,0],[8.999999E+09,8.999999E+09,8.999999E+09,8.999999E+09,8.999999E+09,8.999999E+09]];
	LOCAL CONST Robtarget Tr_meulage_bavure_P125 :=[[-7.749427734375,73.4134375,80.4652421875],[0.167156940708146,-0.147787029239311,0.645668672358269,-0.730294130263159],[0,0,0,0],[8.999999E+09,8.999999E+09,8.999999E+09,8.999999E+09,8.999999E+09,8.999999E+09]];
	LOCAL CONST Robtarget Tr_meulage_bavure_P126 :=[[-6.020064453125,73.152890625,80.4598359375],[0.140413196025701,-0.124023084614873,0.650287743690007,-0.73622568501175],[0,0,0,0],[8.999999E+09,8.999999E+09,8.999999E+09,8.999999E+09,8.999999E+09,8.999999E+09]];
	LOCAL CONST Robtarget Tr_meulage_bavure_P127 :=[[-2.21548828125,72.2306796875,80.5013828125],[0.11961644159201,-0.105560078516953,0.653204120143041,-0.740184675707702],[0,0,0,0],[8.999999E+09,8.999999E+09,8.999999E+09,8.999999E+09,8.999999E+09,8.999999E+09]];
	LOCAL CONST Robtarget Tr_meulage_bavure_P128 :=[[-0.726382263183594,71.6841796875,80.5460390625],[0.10580421640352,-0.0932960699971016,0.65476673016098,-0.742550900739223],[0,0,0,0],[8.999999E+09,8.999999E+09,8.999999E+09,8.999999E+09,8.999999E+09,8.999999E+09]];
	LOCAL CONST Robtarget Tr_meulage_bavure_P129 :=[[1.93069006347656,71.1298125,80.5613203125],[0.0992996520499811,-0.0874981737588407,0.655299491301341,-0.74368422424563],[0,0,0,0],[8.999999E+09,8.999999E+09,8.999999E+09,8.999999E+09,8.999999E+09,8.999999E+09]];
	LOCAL CONST Robtarget Tr_meulage_bavure_P130 :=[[3.57528393554688,70.8820859375,80.5561796875],[0.0998659898341866,-0.0879445586808808,0.655014999946451,-0.743806351490772],[0,0,0,0],[8.999999E+09,8.999999E+09,8.999999E+09,8.999999E+09,8.999999E+09,8.999999E+09]];
	LOCAL CONST Robtarget Tr_meulage_bavure_P131 :=[[5.4122744140625,71.07915625,80.47790625],[0.106993601458947,-0.0941711347451615,0.653948468652526,-0.742990960224059],[0,0,0,0],[8.999999E+09,8.999999E+09,8.999999E+09,8.999999E+09,8.999999E+09,8.999999E+09]];
	LOCAL CONST Robtarget Tr_meulage_bavure_P132 :=[[6.97133837890625,71.2244765625,80.4148359375],[0.119893954377034,-0.10548070550937,0.652059753094324,-0.741159455760805],[0,0,0,0],[8.999999E+09,8.999999E+09,8.999999E+09,8.999999E+09,8.999999E+09,8.999999E+09]];
	LOCAL CONST Robtarget Tr_meulage_bavure_P133 :=[[9.4200693359375,72.1266640625,80.2126171875],[0.137621176675066,-0.121035115778275,0.649221957205297,-0.73818816216574],[0,0,0,0],[8.999999E+09,8.999999E+09,8.999999E+09,8.999999E+09,8.999999E+09,8.999999E+09]];
	LOCAL CONST Robtarget Tr_meulage_bavure_P134 :=[[10.3193076171875,72.291734375,80.163796875],[0.15914116514657,-0.139927241227188,0.645320492387921,-0.733931821644593],[0,0,0,0],[8.999999E+09,8.999999E+09,8.999999E+09,8.999999E+09,8.999999E+09,8.999999E+09]];
	LOCAL CONST Robtarget Tr_meulage_bavure_P135 :=[[12.9175185546875,74.01015625,79.83271875],[0.18330581906679,-0.161146031043023,0.640284028539511,-0.728331858545642],[0,0,0,0],[8.999999E+09,8.999999E+09,8.999999E+09,8.999999E+09,8.999999E+09,8.999999E+09]];
	LOCAL CONST Robtarget Tr_meulage_bavure_P136 :=[[12.9989384765625,74.0414453125,79.825796875],[0.208850960944889,-0.183588303370692,0.634182602594527,-0.721449261933436],[0,0,0,0],[8.999999E+09,8.999999E+09,8.999999E+09,8.999999E+09,8.999999E+09,8.999999E+09]];
	LOCAL CONST Robtarget Tr_meulage_bavure_P137 :=[[13.1842744140625,74.2001171875,79.7966484375],[0.234487873228421,-0.206127349375205,0.627225112555585,-0.713523378263107],[0,0,0,0],[8.999999E+09,8.999999E+09,8.999999E+09,8.999999E+09,8.999999E+09,8.999999E+09]];
	LOCAL CONST Robtarget Tr_meulage_bavure_P138 :=[[16.007322265625,77.160265625,79.269609375],[0.258919773477978,-0.22762500702109,0.619783379239958,-0.704993595643719],[0,0,0,0],[8.999999E+09,8.999999E+09,8.999999E+09,8.999999E+09,8.999999E+09,8.999999E+09]];
	LOCAL CONST Robtarget Tr_meulage_bavure_P139 :=[[16.41192578125,77.7266328125,79.1723125],[0.280873973693305,-0.246963934019434,0.612396593795044,-0.69648333655846],[0,0,0,0],[8.999999E+09,8.999999E+09,8.999999E+09,8.999999E+09,8.999999E+09,8.999999E+09]];
	LOCAL CONST Robtarget Tr_meulage_bavure_P140 :=[[17.965533203125,80.422703125,78.7189375],[0.299266259822404,-0.263199861872182,0.60569505132338,-0.688693722379362],[0,0,0,0],[8.999999E+09,8.999999E+09,8.999999E+09,8.999999E+09,8.999999E+09,8.999999E+09]];
	LOCAL CONST Robtarget Tr_meulage_bavure_P141 :=[[21.11534375,86.9008203125,77.6448203125],[0.313204435681894,-0.275544087648036,0.600307707668791,-0.682355547603183],[0,0,0,0],[8.999999E+09,8.999999E+09,8.999999E+09,8.999999E+09,8.999999E+09,8.999999E+09]];
	LOCAL CONST Robtarget Tr_meulage_bavure_P142 :=[[21.339029296875,87.3939296875,77.563484375],[0.321955731640158,-0.28335178319806,0.596820200445433,-0.67813119834056],[0,0,0,0],[8.999999E+09,8.999999E+09,8.999999E+09,8.999999E+09,8.999999E+09,8.999999E+09]];
	LOCAL CONST Robtarget Tr_meulage_bavure_P143 :=[[21.495451171875,87.7721171875,77.5015],[0.324923595993313,-0.286094433348839,0.595698973068319,-0.67654812501324],[0,0,0,0],[8.999999E+09,8.999999E+09,8.999999E+09,8.999999E+09,8.999999E+09,8.999999E+09]];
	LOCAL CONST Robtarget Tr_meulage_bavure_P144 :=[[23.332166015625,92.6607109375,76.7050859375],[0.321590336041686,-0.283307970635604,0.597245168152768,-0.677948713884099],[0,0,0,0],[8.999999E+09,8.999999E+09,8.999999E+09,8.999999E+09,8.999999E+09,8.999999E+09]];
	LOCAL CONST Robtarget Tr_meulage_bavure_P145 :=[[23.497529296875,93.205125,76.6174140625],[0.311407209768616,-0.274499525637445,0.601586700001717,-0.682472711916006],[0,0,0,0],[8.999999E+09,8.999999E+09,8.999999E+09,8.999999E+09,8.999999E+09,8.999999E+09]];
	LOCAL CONST Robtarget Tr_meulage_bavure_P146 :=[[23.7410703125,94.126109375,76.4700625],[0.293837714569981,-0.259182956580841,0.608608919104422,-0.689984620191532],[0,0,0,0],[8.999999E+09,8.999999E+09,8.999999E+09,8.999999E+09,8.999999E+09,8.999999E+09]];
	LOCAL CONST Robtarget Tr_meulage_bavure_P147 :=[[25.480072265625,98.968515625,75.68328125],[0.268470704011204,-0.236974490494014,0.617875646578929,-0.69999732664311],[0,0,0,0],[8.999999E+09,8.999999E+09,8.999999E+09,8.999999E+09,8.999999E+09,8.999999E+09]];
	LOCAL CONST Robtarget Tr_meulage_bavure_P148 :=[[26.111095703125,100.2981328125,75.4632265625],[0.23519716021745,-0.207761747028165,0.6285976827237,-0.711605442342769],[0,0,0,0],[8.999999E+09,8.999999E+09,8.999999E+09,8.999999E+09,8.999999E+09,8.999999E+09]];
	LOCAL CONST Robtarget Tr_meulage_bavure_P149 :=[[28.573197265625,102.38646875,75.0790859375],[0.194680678621475,-0.172111219310081,0.639591874964701,-0.723463471806433],[0,0,0,0],[8.999999E+09,8.999999E+09,8.999999E+09,8.999999E+09,8.999999E+09,8.999999E+09]];
	LOCAL CONST Robtarget Tr_meulage_bavure_P150 :=[[29.56271484375,103.41746875,74.8953515625],[0.148646099443202,-0.131528281488131,0.649484807452777,-0.734012352196562],[0,0,0,0],[8.999999E+09,8.999999E+09,8.999999E+09,8.999999E+09,8.999999E+09,8.999999E+09]];
	LOCAL CONST Robtarget Tr_meulage_bavure_P151 :=[[31.676603515625,103.3441875,74.85121875],[0.0999512380555259,-0.0885239958546248,0.657081136920145,-0.7419013624956],[0,0,0,0],[8.999999E+09,8.999999E+09,8.999999E+09,8.999999E+09,8.999999E+09,8.999999E+09]];
	LOCAL CONST Robtarget Tr_meulage_bavure_P152 :=[[33.67269140625,103.159265625,74.82725],[0.05199434434757,-0.0460950552500032,0.661777934913066,-0.7464729056701],[0,0,0,0],[8.999999E+09,8.999999E+09,8.999999E+09,8.999999E+09,8.999999E+09,8.999999E+09]];
	LOCAL CONST Robtarget Tr_meulage_bavure_P153 :=[[34.43504296875,102.8518984375,74.8543359375],[0.00778924079640987,-0.00691251890829559,0.66372413595808,-0.747904951285161],[0,0,0,0],[8.999999E+09,8.999999E+09,8.999999E+09,8.999999E+09,8.999999E+09,8.999999E+09]];
	LOCAL CONST Robtarget Tr_meulage_bavure_P154 :=[[37.26056640625,102.0111328125,74.909046875],[0.0306472773472847,-0.0272265431638739,-0.663594552079053,0.746968359563875],[0,0,0,0],[8.999999E+09,8.999999E+09,8.999999E+09,8.999999E+09,8.999999E+09,8.999999E+09]];
	LOCAL CONST Robtarget Tr_meulage_bavure_P155 :=[[37.58883203125,101.817640625,74.9300703125],[0.0625312744147801,-0.0556130546416597,-0.66223102847581,0.744612041802548],[0,0,0,0],[8.999999E+09,8.999999E+09,8.999999E+09,8.999999E+09,8.999999E+09,8.999999E+09]];
	LOCAL CONST Robtarget Tr_meulage_bavure_P156 :=[[41.4956484375,99.9562265625,75.112703125],[0.0879650814804871,-0.078323066120627,-0.660360517041206,0.741654656350694],[0,0,0,0],[8.999999E+09,8.999999E+09,8.999999E+09,8.999999E+09,8.999999E+09,8.999999E+09]];
	LOCAL CONST Robtarget Tr_meulage_bavure_P157 :=[[43.8988984375,98.78621875,75.2288671875],[0.107560795780834,-0.0958865625425415,-0.658492221699123,0.738663953565166],[0,0,0,0],[8.999999E+09,8.999999E+09,8.999999E+09,8.999999E+09,8.999999E+09,8.999999E+09]];
	LOCAL CONST Robtarget Tr_meulage_bavure_P158 :=[[46.93534765625,97.4875234375,75.34815625],[0.122156615317671,-0.109034948301667,-0.656914711635807,0.735970246015033],[0,0,0,0],[8.999999E+09,8.999999E+09,8.999999E+09,8.999999E+09,8.999999E+09,8.999999E+09]];
	LOCAL CONST Robtarget Tr_meulage_bavure_P159 :=[[55.402203125,93.8694296875,75.68028125],[0.132642422226631,-0.118546746465885,-0.655749222770095,0.733720391950927],[0,0,0,0],[8.999999E+09,8.999999E+09,8.999999E+09,8.999999E+09,8.999999E+09,8.999999E+09]];
	LOCAL CONST Robtarget Tr_meulage_bavure_P160 :=[[57.37942578125,93.0266015625,75.757515625],[0.139847413227806,-0.125152335342899,-0.655021919520851,0.731932974335034],[0,0,0,0],[8.999999E+09,8.999999E+09,8.999999E+09,8.999999E+09,8.999999E+09,8.999999E+09]];
	LOCAL CONST Robtarget Tr_meulage_bavure_P161 :=[[58.47840234375,92.57946875,75.7971796875],[0.144524946427824,-0.129515361764061,-0.65468934655818,0.730561544587711],[0,0,0,0],[8.999999E+09,8.999999E+09,8.999999E+09,8.999999E+09,8.999999E+09,8.999999E+09]];
	LOCAL CONST Robtarget Tr_meulage_bavure_P162 :=[[59.01814453125,92.3178125,75.8231015625],[0.147339326326402,-0.132224542671511,-0.654682109724518,0.729519793041728],[0,0,0,0],[8.999999E+09,8.999999E+09,8.999999E+09,8.999999E+09,8.999999E+09,8.999999E+09]];
	LOCAL CONST Robtarget Tr_meulage_bavure_P163 :=[[60.17047265625,91.812859375,75.8702265625],[0.14881257660618,-0.133741554008729,-0.654924409449461,0.728726307801794],[0,0,0,0],[8.999999E+09,8.999999E+09,8.999999E+09,8.999999E+09,8.999999E+09,8.999999E+09]];
	LOCAL CONST Robtarget Tr_meulage_bavure_P164 :=[[69.8240546875,87.62321875,76.2587578125],[0.14939403361211,-0.134465342037131,-0.655341344619923,0.728099043086648],[0,0,0,0],[8.999999E+09,8.999999E+09,8.999999E+09,8.999999E+09,8.999999E+09,8.999999E+09]];
	LOCAL CONST Robtarget Tr_meulage_bavure_P165 :=[[74.1051328125,85.768046875,76.4306328125],[0.149405683276414,-0.134684348303256,-0.655880813436513,0.727570221142051],[0,0,0,0],[8.999999E+09,8.999999E+09,8.999999E+09,8.999999E+09,8.999999E+09,8.999999E+09]];
	LOCAL CONST Robtarget Tr_meulage_bavure_P166 :=[[79.0934453125,83.7188359375,76.6136953125],[0.149085355230857,-0.134607865776139,-0.656491491760993,0.727099168320462],[0,0,0,0],[8.999999E+09,8.999999E+09,8.999999E+09,8.999999E+09,8.999999E+09,8.999999E+09]];
	LOCAL CONST Robtarget Tr_meulage_bavure_P167 :=[[85.848984375,80.8991796875,76.86840625],[0.148606125762516,-0.134393592060356,-0.657148150340182,0.726643578588188],[0,0,0,0],[8.999999E+09,8.999999E+09,8.999999E+09,8.999999E+09,8.999999E+09,8.999999E+09]];
	LOCAL CONST Robtarget Tr_meulage_bavure_P168 :=[[92.480953125,78.1748203125,77.1117734375],[0.148082159529039,-0.134144175550706,-0.657829506437532,0.726179974011395],[0,0,0,0],[8.999999E+09,8.999999E+09,8.999999E+09,8.999999E+09,8.999999E+09,8.999999E+09]];
	LOCAL CONST Robtarget Tr_meulage_bavure_P169 :=[[95.6069375,76.8302109375,77.2357421875],[0.14758749667998,-0.133926738804224,-0.658522311425872,0.725692720654775],[0,0,0,0],[8.999999E+09,8.999999E+09,8.999999E+09,8.999999E+09,8.999999E+09,8.999999E+09]];
	LOCAL CONST Robtarget Tr_meulage_bavure_P170 :=[[100.9483515625,74.641640625,77.4308828125],[0.147138708275564,-0.133756579282908,-0.659223841931464,0.725178118985022],[0,0,0,0],[8.999999E+09,8.999999E+09,8.999999E+09,8.999999E+09,8.999999E+09,8.999999E+09]];
	LOCAL CONST Robtarget Tr_meulage_bavure_P171 :=[[107.37103125,72.1147421875,77.6495],[0.146789819569276,-0.133682764818109,-0.659923266651187,0.724626075568518],[0,0,0,0],[8.999999E+09,8.999999E+09,8.999999E+09,8.999999E+09,8.999999E+09,8.999999E+09]];
	LOCAL CONST Robtarget Tr_meulage_bavure_P172 :=[[108.4919609375,71.6649921875,77.6889921875],[0.146587902527637,-0.133747908239606,-0.660609711408511,0.724029207329954],[0,0,0,0],[8.999999E+09,8.999999E+09,8.999999E+09,8.999999E+09,8.999999E+09,8.999999E+09]];
	LOCAL CONST Robtarget Tr_meulage_bavure_P173 :=[[109.820328125,71.102265625,77.7403515625],[0.146603804183078,-0.134019216098112,-0.661274287025407,0.723368848952274],[0,0,0,0],[8.999999E+09,8.999999E+09,8.999999E+09,8.999999E+09,8.999999E+09,8.999999E+09]];
	LOCAL CONST Robtarget Tr_meulage_bavure_P174 :=[[120.942828125,66.52378125,78.1499453125],[0.146957022088388,-0.134605629321121,-0.661889930349424,0.722624853098765],[0,0,0,0],[8.999999E+09,8.999999E+09,8.999999E+09,8.999999E+09,8.999999E+09,8.999999E+09]];
	LOCAL CONST Robtarget Tr_meulage_bavure_P175 :=[[130.8547421875,62.4051640625,78.52084375],[0.147828897608492,-0.135675246621816,-0.662420918458549,0.721759912487871],[0,0,0,0],[8.999999E+09,8.999999E+09,8.999999E+09,8.999999E+09,8.999999E+09,8.999999E+09]];
	LOCAL CONST Robtarget Tr_meulage_bavure_P176 :=[[132.648171875,61.680234375,78.5848515625],[0.149479321489397,-0.137471794233252,-0.6628193177953,0.72071352852207],[0,0,0,0],[8.999999E+09,8.999999E+09,8.999999E+09,8.999999E+09,8.999999E+09,8.999999E+09]];
	LOCAL CONST Robtarget Tr_meulage_bavure_P177 :=[[137.100265625,60.018421875,78.7226484375],[0.152253990539855,-0.140316650120236,-0.663006397818945,0.719411201271478],[0,0,0,0],[8.999999E+09,8.999999E+09,8.999999E+09,8.999999E+09,8.999999E+09,8.999999E+09]];
	LOCAL CONST Robtarget Tr_meulage_bavure_P178 :=[[146.24603125,56.16858203125,79.07246875],[0.156612365600016,-0.144641954973452,-0.662877145822063,0.717736136299002],[0,0,0,0],[8.999999E+09,8.999999E+09,8.999999E+09,8.999999E+09,8.999999E+09,8.999999E+09]];
	LOCAL CONST Robtarget Tr_meulage_bavure_P179 :=[[148.077671875,55.38012109375,79.1451953125],[0.163073095928608,-0.150939708257558,-0.662295268423289,0.715534308946473],[0,0,0,0],[8.999999E+09,8.999999E+09,8.999999E+09,8.999999E+09,8.999999E+09,8.999999E+09]];
	LOCAL CONST Robtarget Tr_meulage_bavure_P180 :=[[148.886515625,55.048984375,79.174703125],[0.172234737137111,-0.159775795091118,-0.661058787572695,0.712606602550966],[0,0,0,0],[8.999999E+09,8.999999E+09,8.999999E+09,8.999999E+09,8.999999E+09,8.999999E+09]];
	LOCAL CONST Robtarget Tr_meulage_bavure_P181 :=[[154.880796875,52.67449609375,79.3812109375],[0.184731821506807,-0.171760030103712,-0.65890762877984,0.708670150999234],[0,0,0,0],[8.999999E+09,8.999999E+09,8.999999E+09,8.999999E+09,8.999999E+09,8.999999E+09]];
	LOCAL CONST Robtarget Tr_meulage_bavure_P182 :=[[162.227578125,49.7510625,79.636328125],[0.201136568979911,-0.187444925193993,-0.65549458786859,0.703374243140161],[0,0,0,0],[8.999999E+09,8.999999E+09,8.999999E+09,8.999999E+09,8.999999E+09,8.999999E+09]];
	LOCAL CONST Robtarget Tr_meulage_bavure_P183 :=[[166.219328125,48.089078125,79.7862109375],[0.221870160473928,-0.207252178643746,-0.650400786093515,0.696275077672347],[0,0,0,0],[8.999999E+09,8.999999E+09,8.999999E+09,8.999999E+09,8.999999E+09,8.999999E+09]];
	LOCAL CONST Robtarget Tr_meulage_bavure_P184 :=[[169.836046875,46.905375,79.8726953125],[0.247134079302345,-0.231403068777937,-0.643129055871858,0.686849608066357],[0,0,0,0],[8.999999E+09,8.999999E+09,8.999999E+09,8.999999E+09,8.999999E+09,8.999999E+09]];
	LOCAL CONST Robtarget Tr_meulage_bavure_P185 :=[[171.43740625,46.3769765625,79.9116484375],[0.276685600126164,-0.259698005056687,-0.633180916094997,0.674599104910095],[0,0,0,0],[8.999999E+09,8.999999E+09,8.999999E+09,8.999999E+09,8.999999E+09,8.999999E+09]];
	LOCAL CONST Robtarget Tr_meulage_bavure_P186 :=[[175.519234375,44.64690234375,80.0695859375],[0.309782204462912,-0.291477484410174,-0.620181518750722,0.659128777766579],[0,0,0,0],[8.999999E+09,8.999999E+09,8.999999E+09,8.999999E+09,8.999999E+09,8.999999E+09]];
	LOCAL CONST Robtarget Tr_meulage_bavure_P187 :=[[176.500171875,43.8523203125,80.16553125],[0.345199523569393,-0.325609018471639,-0.60398620622411,0.640325478728128],[0,0,0,0],[8.999999E+09,8.999999E+09,8.999999E+09,8.999999E+09,8.999999E+09,8.999999E+09]];
	LOCAL CONST Robtarget Tr_meulage_bavure_P188 :=[[176.789203125,43.49858984375,80.212109375],[0.381293435737265,-0.360558299958492,-0.584866667864363,0.618501421999942],[0,0,0,0],[8.999999E+09,8.999999E+09,8.999999E+09,8.999999E+09,8.999999E+09,8.999999E+09]];
	LOCAL CONST Robtarget Tr_meulage_bavure_P189 :=[[177.998515625,41.684828125,80.4580859375],[0.416352510116684,-0.394698207475455,-0.563500905268504,0.594416219577474],[0,0,0,0],[8.999999E+09,8.999999E+09,8.999999E+09,8.999999E+09,8.999999E+09,8.999999E+09]];
	LOCAL CONST Robtarget Tr_meulage_bavure_P190 :=[[178.200265625,40.82044140625,80.5851171875],[0.448873436158103,-0.426608356985801,-0.540915840329414,0.569146731293624],[0,0,0,0],[8.999999E+09,8.999999E+09,8.999999E+09,8.999999E+09,8.999999E+09,8.999999E+09]];
	LOCAL CONST Robtarget Tr_meulage_bavure_P191 :=[[178.205,40.14398828125,80.6885390625],[0.47791109401537,-0.455366011554948,-0.518168875365487,0.543823315370018],[0,0,0,0],[8.999999E+09,8.999999E+09,8.999999E+09,8.999999E+09,8.999999E+09,8.999999E+09]];
	LOCAL CONST Robtarget Tr_meulage_bavure_P192 :=[[178.05775,38.57928515625,80.93190625],[0.502934785531011,-0.480432030303729,-0.496299971958842,0.519545959078469],[0,0,0,0],[8.999999E+09,8.999999E+09,8.999999E+09,8.999999E+09,8.999999E+09,8.999999E+09]];
	LOCAL CONST Robtarget Tr_meulage_bavure_P193 :=[[177.7885625,37.72346484375,81.0699609375],[0.523784569081067,-0.50163235848101,-0.476205763057921,0.497235128835207],[0,0,0,0],[8.999999E+09,8.999999E+09,8.999999E+09,8.999999E+09,8.999999E+09,8.999999E+09]];
	LOCAL CONST Robtarget Tr_meulage_bavure_P194 :=[[175.946046875,33.9934140625,81.6891875],[0.540563216894635,-0.519031014796201,-0.458578255799512,0.477602551844132],[0,0,0,0],[8.999999E+09,8.999999E+09,8.999999E+09,8.999999E+09,8.999999E+09,8.999999E+09]];
	LOCAL CONST Robtarget Tr_meulage_bavure_P195 :=[[175.689703125,33.4522578125,81.778734375],[0.553490404830816,-0.532808836155291,-0.443940408941852,0.461172450590455],[0,0,0,0],[8.999999E+09,8.999999E+09,8.999999E+09,8.999999E+09,8.999999E+09,8.999999E+09]];
	LOCAL CONST Robtarget Tr_meulage_bavure_P196 :=[[175.6156875,33.317203125,81.80134375],[0.562862949734296,-0.543218902687694,-0.432618531378649,0.448263014185831],[0,0,0,0],[8.999999E+09,8.999999E+09,8.999999E+09,8.999999E+09,8.999999E+09,8.999999E+09]];
	LOCAL CONST Robtarget Tr_meulage_bavure_P197 :=[[175.14046875,32.3669609375,81.95925],[0.568962230507439,-0.550509997156796,-0.424806125785407,0.439044962141257],[0,0,0,0],[8.999999E+09,8.999999E+09,8.999999E+09,8.999999E+09,8.999999E+09,8.999999E+09]];
	LOCAL CONST Robtarget Tr_meulage_bavure_P198 :=[[173.82146875,29.69873828125,82.40221875],[0.572112599941187,-0.5549623045976,-0.420480345561099,0.43347467337905],[0,0,0,0],[8.999999E+09,8.999999E+09,8.999999E+09,8.999999E+09,8.999999E+09,8.999999E+09]];
	LOCAL CONST Robtarget Tr_meulage_bavure_P199 :=[[171.182875,23.856705078125,83.365578125],[0.572639018270833,-0.556871263527351,-0.419448805716341,0.431325457160139],[0,0,0,0],[8.999999E+09,8.999999E+09,8.999999E+09,8.999999E+09,8.999999E+09,8.999999E+09]];
	LOCAL CONST Robtarget Tr_meulage_bavure_P200 :=[[169.290953125,19.605080078125,84.0659296875],[0.570974872685308,-0.556633049978841,-0.421239720491296,0.432093092184618],[0,0,0,0],[8.999999E+09,8.999999E+09,8.999999E+09,8.999999E+09,8.999999E+09,8.999999E+09]];
	LOCAL CONST Robtarget Tr_meulage_bavure_P201 :=[[168.8690625,18.655740234375,84.222296875],[0.567680588447906,-0.554782586380469,-0.425119979418959,0.435003487856432],[0,0,0,0],[8.999999E+09,8.999999E+09,8.999999E+09,8.999999E+09,8.999999E+09,8.999999E+09]];
	LOCAL CONST Robtarget Tr_meulage_bavure_P202 :=[[168.730953125,18.283849609375,84.28284375],[0.563464643178453,-0.552002634439337,-0.430137947923896,0.439069508410264],[0,0,0,0],[8.999999E+09,8.999999E+09,8.999999E+09,8.999999E+09,8.999999E+09,8.999999E+09]];
	LOCAL CONST Robtarget Tr_meulage_bavure_P203 :=[[168.559296875,17.87801953125,84.3494609375],[0.559188096861995,-0.549118026078472,-0.435182883686709,0.443163540365928],[0,0,0,0],[8.999999E+09,8.999999E+09,8.999999E+09,8.999999E+09,8.999999E+09,8.999999E+09]];
	LOCAL CONST Robtarget Tr_meulage_bavure_P204 :=[[168.30575,17.429654296875,84.424734375],[0.555759753198534,-0.547032332664584,-0.439138009726829,0.446144071077279],[0,0,0,0],[8.999999E+09,8.999999E+09,8.999999E+09,8.999999E+09,8.999999E+09,8.999999E+09]];
	LOCAL CONST Robtarget Tr_meulage_bavure_P205 :=[[168.3355625,17.405251953125,84.4276875],[0.553962875504314,-0.546513707951123,-0.441082803335714,0.447094911831944],[0,0,0,0],[8.999999E+09,8.999999E+09,8.999999E+09,8.999999E+09,8.999999E+09,8.999999E+09]];
	LOCAL CONST Robtarget Tr_meulage_bavure_P206 :=[[166.760453125,13.69655859375,85.036640625],[0.554190168326781,-0.54797258176633,-0.440550756691223,0.445549478443268],[0,0,0,0],[8.999999E+09,8.999999E+09,8.999999E+09,8.999999E+09,8.999999E+09,8.999999E+09]];
	LOCAL CONST Robtarget Tr_meulage_bavure_P207 :=[[166.404171875,12.847583984375,85.175921875],[0.556449797438073,-0.551414831162802,-0.437489461807154,0.441484176061286],[0,0,0,0],[8.999999E+09,8.999999E+09,8.999999E+09,8.999999E+09,8.999999E+09,8.999999E+09]];
	LOCAL CONST Robtarget Tr_meulage_bavure_P208 :=[[166.069671875,11.906060546875,85.3288046875],[0.560328136184921,-0.556451564279155,-0.432308330796512,0.43532004724656],[0,0,0,0],[8.999999E+09,8.999999E+09,8.999999E+09,8.999999E+09,8.999999E+09,8.999999E+09]];
	LOCAL CONST Robtarget Tr_meulage_bavure_P209 :=[[164.246640625,7.531775390625,86.0461328125],[0.565198450379859,-0.562453603592058,-0.42568983142573,0.427767253205814],[0,0,0,0],[8.999999E+09,8.999999E+09,8.999999E+09,8.999999E+09,8.999999E+09,8.999999E+09]];
	LOCAL CONST Robtarget Tr_meulage_bavure_P210 :=[[163.41615625,5.710326171875,86.3466953125],[0.570389993215023,-0.568765379239463,-0.418425369282673,0.419620554024007],[0,0,0,0],[8.999999E+09,8.999999E+09,8.999999E+09,8.999999E+09,8.999999E+09,8.999999E+09]];
	LOCAL CONST Robtarget Tr_meulage_bavure_P211 :=[[162.322421875,3.484796875,86.7160078125],[0.575351598083274,-0.574831040108955,-0.411237994584488,0.41161040526256],[0,0,0,0],[8.999999E+09,8.999999E+09,8.999999E+09,8.999999E+09,8.999999E+09,8.999999E+09]];
	LOCAL CONST Robtarget Tr_meulage_bavure_P212 :=[[159.9765,-1.43592248535156,87.530671875],[0.57968639261451,-0.580247081317463,-0.404718055640747,0.404326979409629],[0,0,0,0],[8.999999E+09,8.999999E+09,8.999999E+09,8.999999E+09,8.999999E+09,8.999999E+09]];
	LOCAL CONST Robtarget Tr_meulage_bavure_P213 :=[[158.443734375,-4.93553125,88.1065078125],[0.583179374550334,-0.584786919797512,-0.399250070169675,0.398152554936333],[0,0,0,0],[8.999999E+09,8.999999E+09,8.999999E+09,8.999999E+09,8.999999E+09,8.999999E+09]];
	LOCAL CONST Robtarget Tr_meulage_bavure_P214 :=[[156.827125,-8.6111005859375,88.71146875],[0.585786309919476,-0.588406189620203,-0.394980205998494,0.393221555865068],[0,0,0,0],[8.999999E+09,8.999999E+09,8.999999E+09,8.999999E+09,8.999999E+09,8.999999E+09]];
	LOCAL CONST Robtarget Tr_meulage_bavure_P215 :=[[155.373859375,-11.8955927734375,89.252296875],[0.587559067939165,-0.591151199445424,-0.391902719106949,0.389521321410364],[0,0,0,0],[8.999999E+09,8.999999E+09,8.999999E+09,8.999999E+09,8.999999E+09,8.999999E+09]];
	LOCAL CONST Robtarget Tr_meulage_bavure_P216 :=[[154.1465,-14.60637890625,89.699390625],[0.588621760937856,-0.593141568680219,-0.389881589431515,0.386910646372444],[0,0,0,0],[8.999999E+09,8.999999E+09,8.999999E+09,8.999999E+09,8.999999E+09,8.999999E+09]];
	LOCAL CONST Robtarget Tr_meulage_bavure_P217 :=[[151.75665625,-19.6683984375,90.536828125],[0.589108881764299,-0.594505723980725,-0.388744745677631,0.385215773675749],[0,0,0,0],[8.999999E+09,8.999999E+09,8.999999E+09,8.999999E+09,8.999999E+09,8.999999E+09]];
	LOCAL CONST Robtarget Tr_meulage_bavure_P218 :=[[151.61971875,-19.968552734375,90.5863671875],[0.58918919666911,-0.595403159861753,-0.388253252662106,0.384201222736658],[0,0,0,0],[8.999999E+09,8.999999E+09,8.999999E+09,8.999999E+09,8.999999E+09,8.999999E+09]];
	LOCAL CONST Robtarget Tr_meulage_bavure_P219 :=[[149.3975625,-24.21451171875,91.2945],[0.58899517881961,-0.59597372452971,-0.388206566245175,0.383660867070869],[0,0,0,0],[8.999999E+09,8.999999E+09,8.999999E+09,8.999999E+09,8.999999E+09,8.999999E+09]];
	LOCAL CONST Robtarget Tr_meulage_bavure_P220 :=[[145.75140625,-32.75704296875,92.6976171875],[0.588653852400458,-0.596327051416044,-0.388418786911726,0.383420833781328],[0,0,0,0],[8.999999E+09,8.999999E+09,8.999999E+09,8.999999E+09,8.999999E+09,8.999999E+09]];
	LOCAL CONST Robtarget Tr_meulage_bavure_P221 :=[[145.498140625,-33.32332421875,92.7909296875],[0.588248417785142,-0.596573353996464,-0.388749541278257,0.383324701044207],[0,0,0,0],[8.999999E+09,8.999999E+09,8.999999E+09,8.999999E+09,8.999999E+09,8.999999E+09]];
	LOCAL CONST Robtarget Tr_meulage_bavure_P222 :=[[143.93496875,-37.18019921875,93.42225],[0.587832425160401,-0.596741859199769,-0.389127151197783,0.383317431914519],[0,0,0,0],[8.999999E+09,8.999999E+09,8.999999E+09,8.999999E+09,8.999999E+09,8.999999E+09]];
	LOCAL CONST Robtarget Tr_meulage_bavure_P223 :=[[143.203,-39.1047890625,93.7360234375],[0.587444714822763,-0.596887929651251,-0.389483941404057,0.383322013262749],[0,0,0,0],[8.999999E+09,8.999999E+09,8.999999E+09,8.999999E+09,8.999999E+09,8.999999E+09]];
	LOCAL CONST Robtarget Tr_meulage_bavure_P224 :=[[141.298234375,-43.5161875,94.461171875],[0.587089338471983,-0.597002994254071,-0.389819452050276,0.383346225111746],[0,0,0,0],[8.999999E+09,8.999999E+09,8.999999E+09,8.999999E+09,8.999999E+09,8.999999E+09]];
	LOCAL CONST Robtarget Tr_meulage_bavure_P225 :=[[140.240921875,-46.2259375,94.9036484375],[0.586748361139484,-0.597069081404829,-0.390161528370779,0.383417337257851],[0,0,0,0],[8.999999E+09,8.999999E+09,8.999999E+09,8.999999E+09,8.999999E+09,8.999999E+09]];
	LOCAL CONST Robtarget Tr_meulage_bavure_P226 :=[[140.02446875,-46.67600390625,94.9782109375],[0.586390600920366,-0.597052134860835,-0.390559766542899,0.383585557820323],[0,0,0,0],[8.999999E+09,8.999999E+09,8.999999E+09,8.999999E+09,8.999999E+09,8.999999E+09]];
	LOCAL CONST Robtarget Tr_meulage_bavure_P227 :=[[139.630203125,-47.54828125,95.1220546875],[0.5859785171592,-0.596920295090231,-0.391069481586767,0.383901028012109],[0,0,0,0],[8.999999E+09,8.999999E+09,8.999999E+09,8.999999E+09,8.999999E+09,8.999999E+09]];
	LOCAL CONST Robtarget Tr_meulage_bavure_P228 :=[[138.1680625,-50.71637890625,95.645296875],[0.58550761580572,-0.596663330367305,-0.391699711451848,0.384376167415511],[0,0,0,0],[8.999999E+09,8.999999E+09,8.999999E+09,8.999999E+09,8.999999E+09,8.999999E+09]];
	LOCAL CONST Robtarget Tr_meulage_bavure_P229 :=[[136.613203125,-54.3635,96.244296875],[0.584969017490134,-0.596278963601722,-0.392460308618177,0.385016301345813],[0,0,0,0],[8.999999E+09,8.999999E+09,8.999999E+09,8.999999E+09,8.999999E+09,8.999999E+09]];
	LOCAL CONST Robtarget Tr_meulage_bavure_P230 :=[[134.772640625,-58.42887890625,96.914796875],[0.58437109336419,-0.595770426454938,-0.393339536695556,0.385813469275202],[0,0,0,0],[8.999999E+09,8.999999E+09,8.999999E+09,8.999999E+09,8.999999E+09,8.999999E+09]];
	LOCAL CONST Robtarget Tr_meulage_bavure_P231 :=[[134.5958125,-58.85360546875,96.9844375],[0.583734768559282,-0.595154252506059,-0.394305916416871,0.386740197002649],[0,0,0,0],[8.999999E+09,8.999999E+09,8.999999E+09,8.999999E+09,8.999999E+09,8.999999E+09]];
	LOCAL CONST Robtarget Tr_meulage_bavure_P232 :=[[133.4118125,-61.10366015625,97.3598671875],[0.583080868189484,-0.594462643875666,-0.395321333170207,0.387752381976283],[0,0,0,0],[8.999999E+09,8.999999E+09,8.999999E+09,8.999999E+09,8.999999E+09,8.999999E+09]];
	LOCAL CONST Robtarget Tr_meulage_bavure_P233 :=[[131.89259375,-64.8865625,97.9787109375],[0.582437009176522,-0.593719505964006,-0.396344482435407,0.388812718184957],[0,0,0,0],[8.999999E+09,8.999999E+09,8.999999E+09,8.999999E+09,8.999999E+09,8.999999E+09]];
	LOCAL CONST Robtarget Tr_meulage_bavure_P234 :=[[131.129078125,-66.61509375,98.2633046875],[0.581828734056408,-0.592957006685153,-0.397333280705902,0.389876360520596],[0,0,0,0],[8.999999E+09,8.999999E+09,8.999999E+09,8.999999E+09,8.999999E+09,8.999999E+09]];
	LOCAL CONST Robtarget Tr_meulage_bavure_P235 :=[[130.25046875,-68.928109375,98.6403671875],[0.58128081728044,-0.592189907415536,-0.398254619094211,0.390918128752156],[0,0,0,0],[8.999999E+09,8.999999E+09,8.999999E+09,8.999999E+09,8.999999E+09,8.999999E+09]];
	LOCAL CONST Robtarget Tr_meulage_bavure_P236 :=[[129.1794375,-71.8407265625,99.1142578125],[0.580802820076724,-0.591442560523211,-0.399088118671148,0.391908733416591],[0,0,0,0],[8.999999E+09,8.999999E+09,8.999999E+09,8.999999E+09,8.999999E+09,8.999999E+09]];
	LOCAL CONST Robtarget Tr_meulage_bavure_P237 :=[[128.21934375,-74.0396796875,99.4760078125],[0.580414733445091,-0.59071798084274,-0.399811534694458,0.392838059554064],[0,0,0,0],[8.999999E+09,8.999999E+09,8.999999E+09,8.999999E+09,8.999999E+09,8.999999E+09]];
	LOCAL CONST Robtarget Tr_meulage_bavure_P238 :=[[126.28740625,-78.310671875,100.180375],[0.58011457319909,-0.590030400618924,-0.400421695267385,0.393692359929301],[0,0,0,0],[8.999999E+09,8.999999E+09,8.999999E+09,8.999999E+09,8.999999E+09,8.999999E+09]];
	LOCAL CONST Robtarget Tr_meulage_bavure_P239 :=[[125.6191640625,-80.058875,100.4654765625],[0.579921308050725,-0.589385536407792,-0.400896543362094,0.39445903141183],[0,0,0,0],[8.999999E+09,8.999999E+09,8.999999E+09,8.999999E+09,8.999999E+09,8.999999E+09]];
	LOCAL CONST Robtarget Tr_meulage_bavure_P240 :=[[123.9358125,-84.2095546875,101.1449140625],[0.579832320239363,-0.588810315043412,-0.401228578276745,0.395110770896386],[0,0,0,0],[8.999999E+09,8.999999E+09,8.999999E+09,8.999999E+09,8.999999E+09,8.999999E+09]];
	LOCAL CONST Robtarget Tr_meulage_bavure_P241 :=[[123.06471875,-86.024671875,101.4455703125],[0.579876313015635,-0.588302268465586,-0.401388796326644,0.39563990787721],[0,0,0,0],[8.999999E+09,8.999999E+09,8.999999E+09,8.999999E+09,8.999999E+09,8.999999E+09]];
	LOCAL CONST Robtarget Tr_meulage_bavure_P242 :=[[122.160703125,-87.9678984375,101.766703125],[0.580049492355018,-0.587892138315814,-0.40136948147152,0.396015100051032],[0,0,0,0],[8.999999E+09,8.999999E+09,8.999999E+09,8.999999E+09,8.999999E+09,8.999999E+09]];
	LOCAL CONST Robtarget Tr_meulage_bavure_P243 :=[[121.1965390625,-90.5524921875,102.1875859375],[0.58037124054514,-0.587576276250998,-0.401151912596689,0.396232868090376],[0,0,0,0],[8.999999E+09,8.999999E+09,8.999999E+09,8.999999E+09,8.999999E+09,8.999999E+09]];
	LOCAL CONST Robtarget Tr_meulage_bavure_P244 :=[[119.7116171875,-93.42575,102.6662890625],[0.580826489288309,-0.587360098250536,-0.400750408425359,0.396292586949398],[0,0,0,0],[8.999999E+09,8.999999E+09,8.999999E+09,8.999999E+09,8.999999E+09,8.999999E+09]];
	LOCAL CONST Robtarget Tr_meulage_bavure_P245 :=[[119.5134140625,-93.798046875,102.72846875],[0.581411701957101,-0.587225610234313,-0.400176093993689,0.396214095292229],[0,0,0,0],[8.999999E+09,8.999999E+09,8.999999E+09,8.999999E+09,8.999999E+09,8.999999E+09]];
	LOCAL CONST Robtarget Tr_meulage_bavure_P246 :=[[118.6087578125,-96.2517265625,103.12775],[0.582095012994809,-0.587155751714177,-0.39946993818042,0.396026877327365],[0,0,0,0],[8.999999E+09,8.999999E+09,8.999999E+09,8.999999E+09,8.999999E+09,8.999999E+09]];
	LOCAL CONST Robtarget Tr_meulage_bavure_P247 :=[[118.429390625,-96.4685625,103.165640625],[0.582844985206932,-0.587117757305159,-0.398678753645889,0.395777353656639],[0,0,0,0],[8.999999E+09,8.999999E+09,8.999999E+09,8.999999E+09,8.999999E+09,8.999999E+09]];
	LOCAL CONST Robtarget Tr_meulage_bavure_P248 :=[[118.174625,-97.131359375,103.2737734375],[0.583628738446557,-0.587077497699551,-0.397851562040127,0.395514401680071],[0,0,0,0],[8.999999E+09,8.999999E+09,8.999999E+09,8.999999E+09,8.999999E+09,8.999999E+09]];
	LOCAL CONST Robtarget Tr_meulage_bavure_P249 :=[[115.93303125,-101.9454921875,104.0693828125],[0.584413011371433,-0.587001533663894,-0.397037692539653,0.395286860797066],[0,0,0,0],[8.999999E+09,8.999999E+09,8.999999E+09,8.999999E+09,8.999999E+09,8.999999E+09]];
	LOCAL CONST Robtarget Tr_meulage_bavure_P250 :=[[115.2984609375,-103.450328125,104.3163515625],[0.585172277949434,-0.586877830218657,-0.396269600748265,0.395117983696164],[0,0,0,0],[8.999999E+09,8.999999E+09,8.999999E+09,8.999999E+09,8.999999E+09,8.999999E+09]];
	LOCAL CONST Robtarget Tr_meulage_bavure_P251 :=[[114.8301328125,-104.625359375,104.508484375],[0.585894228581778,-0.58670046513076,-0.395563054583082,0.395019476708193],[0,0,0,0],[8.999999E+09,8.999999E+09,8.999999E+09,8.999999E+09,8.999999E+09,8.999999E+09]];
	LOCAL CONST Robtarget Tr_meulage_bavure_P252 :=[[113.4772265625,-107.830765625,105.034578125],[0.58658667666346,-0.586471808603993,-0.394908718391514,0.394986066351779],[0,0,0,0],[8.999999E+09,8.999999E+09,8.999999E+09,8.999999E+09,8.999999E+09,8.999999E+09]];
	LOCAL CONST Robtarget Tr_meulage_bavure_P253 :=[[112.65996875,-109.8169453125,105.3600078125],[0.587264832205362,-0.586212399632958,-0.394281845447532,0.394989703311194],[0,0,0,0],[8.999999E+09,8.999999E+09,8.999999E+09,8.999999E+09,8.999999E+09,8.999999E+09]];
